(* CoDeSys 2.3.9.48 project: RCS_FB-20170118.pro *)
(* Libraries: WagoLibTerminalDiag.lib 8.11.10 11:37:48, C:\Program Files (x86)\WAGO Software\CoDeSys V2.3\Targets\WAGO\Libraries\32_Bit\SysLibMem.lib 8.11.10 11:37:48, C:\Program Files (x86)\WAGO Software\CoDeSys V2.3\Targets\WAGO\Libraries\32_Bit\SysLibRtc.lib 8.11.10 11:37:48, Util.lib 26.9.14 10:12:46, C:\Program Files (x86)\WAGO Software\CoDeSys V2.3\Targets\WAGO\Libraries\Application\WagoLib_CAN_Gateway_02.lib 25.11.15 11:32:40, C:\Program Files (x86)\WAGO Software\CoDeSys V2.3\Targets\WAGO\Libraries\Application\WagoLibMBX_System_01.lib 22.10.13 15:28:54, C:\Program Files (x86)\WAGO Software\CoDeSys V2.3\Targets\WAGO\Libraries\Application\WagoLibMBX_01.lib 20.3.12 15:32:38, Standard.lib 8.11.10 11:37:48, SYSLIBCALLBACK.LIB 8.11.10 11:37:48, WagoLibModbus_IP_01.lib 12.2.16 10:20:24, SysLibSockets.lib 5.5.11 08:22:24, Wago_MBCFG_ETHERNET_01.lib 1.4.15 13:24:28, Wago_MBCFG_COMMON_01.lib 1.4.15 13:24:28 *)

(* PLC configuration (modules and I/O channels)
0750-0658#48 CAN Gateway (48 Bytes) [Type_33_1_Channels] node 0, in %IB106 out %QB134 {INTTypePAAssignment = PLC; INTTypeModule = plugged}
  AT %IB0 [BYTEOnB_I] First Byte of 48
  AT %QB0 [BYTEOnB_Q] First Byte of 48
0750-0658#48 CAN Gateway (48 Bytes) [Type_33_1_Channels] node 1, in %IB106 out %QB134 {INTTypePAAssignment = PLC; INTTypeModule = plugged}
  AT %IB48 [BYTEOnB_I] First Byte of 48
  AT %QB48 [BYTEOnB_Q] First Byte of 48
AT %IX48.0 [BOOLOnX_I] moving negative
AT %IX48.1 [BOOLOnX_I] moving positive
AT %IX48.2 [BOOLOnX_I] On target
AT %IX48.3 [BOOLOnX_I] busy
AT %IX48.4 [BOOLOnX_I] standstill
AT %IX48.5 [BOOLOnX_I] reference ok
AT %IX48.6 [BOOLOnX_I] error, see extended info
AT %IX48.8 [BOOLOnX_I] preset input enabled
AT %IX48.9 [BOOLOnX_I] optimize on (and Z-Input for 750-636 > FW2)
AT %IX48.10 [BOOLOnX_I] extended info on
AT %IX48.11 [BOOLOnX_I] PWM active
AT %IX48.12 [BOOLOnX_I] current control on
AT %IX48.13 [BOOLOnX_I] preset input
AT %IX48.14 [BOOLOnX_I] limit switch negative
AT %IX48.15 [BOOLOnX_I] limit switch positive
AT %IW49 [WORDOnW_I] actual position low word
AT %IX49.0 [BOOLOnX_I] over temperature warning
AT %IX49.1 [BOOLOnX_I] over temperature
AT %IX49.2 [BOOLOnX_I] overflow warning
AT %IX49.3 [BOOLOnX_I] 24V ok
AT %IX49.4 [BOOLOnX_I] overload
AT %IX49.5 [BOOLOnX_I] motion detection timeout
AT %IX49.6 [BOOLOnX_I] parameter write failed
AT %IX49.7 [BOOLOnX_I] 24VL Ok (only 750-636/000-800)
AT %IX49.8 [BOOLOnX_I] 24VM Ok (only 750-636/000-800)
AT %IW50 [WORDOnW_I] actual position high word
AT %QX48.0 [BOOLOnX_Q] move negative
AT %QX48.1 [BOOLOnX_Q] move positive
AT %QX48.2 [BOOLOnX_Q] positioning
AT %QX48.3 [BOOLOnX_Q] preset
AT %QX48.4 [BOOLOnX_Q] current control on
AT %QX48.8 [BOOLOnX_Q] preset input enable
AT %QX48.9 [BOOLOnX_Q] optimize on
AT %QX48.10 [BOOLOnX_Q] extended info on
AT %QX48.15 [BOOLOnX_Q] error quit
AT %QW49 [WORDOnW_Q] target position low word
AT %QW50 [WORDOnW_Q] target position high word
0753-0430 8 DI 24 V DC 3.0ms [Type_1_8_Channels] node 3, in %IB110 out %QB134 {INTTypePAAssignment = PLC; INTTypeModule = plugged}
  AT %IX55.0 [BOOLOnX_I] Ch_1 Digital input
  AT %IX55.1 [BOOLOnX_I] Ch_2 Digital input
  AT %IX55.2 [BOOLOnX_I] Ch_3 Digital input
  AT %IX55.3 [BOOLOnX_I] Ch_4 Digital input
  AT %IX55.4 [BOOLOnX_I] Ch_5 Digital input
  AT %IX55.5 [BOOLOnX_I] Ch_6 Digital input
  AT %IX55.6 [BOOLOnX_I] Ch_7 Digital input
  AT %IX55.7 [BOOLOnX_I] Ch_8 Digital input
  AT %IX55.8 [BOOLOnX_I] Ch_1 Digital input
  AT %IX55.9 [BOOLOnX_I] Ch_2 Digital input
  AT %IX55.10 [BOOLOnX_I] Ch_3 Digital input
  AT %IX55.11 [BOOLOnX_I] Ch_4 Digital input
  AT %IX55.12 [BOOLOnX_I] Ch_5 Digital input
  AT %IX55.13 [BOOLOnX_I] Ch_6 Digital input
  AT %IX55.14 [BOOLOnX_I] Ch_7 Digital input
  AT %IX55.15 [BOOLOnX_I] Ch_8 Digital input
  AT %IX56.0 [BOOLOnX_I] Ch_1 Digital input
  AT %IX56.1 [BOOLOnX_I] Ch_2 Digital input
  AT %IX56.2 [BOOLOnX_I] Ch_3 Digital input
  AT %IX56.3 [BOOLOnX_I] Ch_4 Digital input
  AT %IX56.4 [BOOLOnX_I] Ch_5 Digital input
  AT %IX56.5 [BOOLOnX_I] Ch_6 Digital input
  AT %IX56.6 [BOOLOnX_I] Ch_7 Digital input
  AT %IX56.7 [BOOLOnX_I] Ch_8 Digital input
  AT %IX56.8 [BOOLOnX_I] Ch_1 Digital input
  AT %IX56.9 [BOOLOnX_I] Ch_2 Digital input
  AT %IX56.10 [BOOLOnX_I] Ch_3 Digital input
  AT %IX56.11 [BOOLOnX_I] Ch_4 Digital input
  AT %IX56.12 [BOOLOnX_I] Ch_5 Digital input
  AT %IX56.13 [BOOLOnX_I] Ch_6 Digital input
  AT %IX56.14 [BOOLOnX_I] Ch_7 Digital input
  AT %IX56.15 [BOOLOnX_I] Ch_8 Digital input
0753-0530 8 DO 24 V DC 0.5A [Type_10_8_Channels] node 7, in %IB113 out %QB134 {INTTypePAAssignment = PLC; INTTypeModule = plugged}
  AT %QX67.0 [BOOLOnX_Q] Ch_1 Digital output
  AT %QX67.1 [BOOLOnX_Q] Ch_2 Digital output
  AT %QX67.2 [BOOLOnX_Q] Ch_3 Digital output
  AT %QX67.3 [BOOLOnX_Q] Ch_4 Digital output
  AT %QX67.4 [BOOLOnX_Q] Ch_5 Digital output
  AT %QX67.5 [BOOLOnX_Q] Ch_6 Digital output
  AT %QX67.6 [BOOLOnX_Q] Ch_7 Digital output
  AT %QX67.7 [BOOLOnX_Q] Ch_8 Digital output
0753-0530 8 DO 24 V DC 0.5A [Type_10_8_Channels] node 8, in %IB114 out %QB134 {INTTypePAAssignment = PLC; INTTypeModule = plugged}
  AT %QX67.8 [BOOLOnX_Q] Ch_1 Digital output
  AT %QX67.9 [BOOLOnX_Q] Ch_2 Digital output
  AT %QX67.10 [BOOLOnX_Q] Ch_3 Digital output
  AT %QX67.11 [BOOLOnX_Q] Ch_4 Digital output
  AT %QX67.12 [BOOLOnX_Q] Ch_5 Digital output
  AT %QX67.13 [BOOLOnX_Q] Ch_6 Digital output
  AT %QX67.14 [BOOLOnX_Q] Ch_7 Digital output
  AT %QX67.15 [BOOLOnX_Q] Ch_8 Digital output
0753-0530 8 DO 24 V DC 0.5A [Type_10_8_Channels] node 9, in %IB114 out %QB135 {INTTypePAAssignment = PLC; INTTypeModule = plugged}
  AT %QX68.0 [BOOLOnX_Q] Ch_1 Digital output
  AT %QX68.1 [BOOLOnX_Q] Ch_2 Digital output
  AT %QX68.2 [BOOLOnX_Q] Ch_3 Digital output
  AT %QX68.3 [BOOLOnX_Q] Ch_4 Digital output
  AT %QX68.4 [BOOLOnX_Q] Ch_5 Digital output
  AT %QX68.5 [BOOLOnX_Q] Ch_6 Digital output
  AT %QX68.6 [BOOLOnX_Q] Ch_7 Digital output
  AT %QX68.7 [BOOLOnX_Q] Ch_8 Digital output
  AT %QX68.8 [BOOLOnX_Q] Ch_1 Digital output
  AT %QX68.9 [BOOLOnX_Q] Ch_2 Digital output
  AT %QX68.10 [BOOLOnX_Q] Ch_3 Digital output
  AT %QX68.11 [BOOLOnX_Q] Ch_4 Digital output
  AT %QX68.12 [BOOLOnX_Q] Ch_5 Digital output
  AT %QX68.13 [BOOLOnX_Q] Ch_6 Digital output
  AT %QX68.14 [BOOLOnX_Q] Ch_7 Digital output
  AT %QX68.15 [BOOLOnX_Q] Ch_8 Digital output
  AT %QX69.0 [BOOLOnX_Q] Ch_1 Digital output
  AT %QX69.1 [BOOLOnX_Q] Ch_2 Digital output
  AT %QX69.2 [BOOLOnX_Q] Ch_3 Digital output
  AT %QX69.3 [BOOLOnX_Q] Ch_4 Digital output
  AT %QX69.4 [BOOLOnX_Q] Ch_5 Digital output
  AT %QX69.5 [BOOLOnX_Q] Ch_6 Digital output
  AT %QX69.6 [BOOLOnX_Q] Ch_7 Digital output
  AT %QX69.7 [BOOLOnX_Q] Ch_8 Digital output
0753-0555 4 AO 4-20mA [Type_14_4_Channels] node 12, in %IB202 out %QB230 {INTTypePAAssignment = PLC; INTTypeModule = plugged}
  AT %QW51 [WORDOnW_Q] Ch_1 Analog output
  AT %QW52 [WORDOnW_Q] Ch_2 Analog output
  AT %QW53 [WORDOnW_Q] Ch_3 Analog output
  AT %QW54 [WORDOnW_Q] Ch_4 Analog output
0753-0555 4 AO 4-20mA [Type_14_4_Channels] node 13, in %IB208 out %QB236 {INTTypePAAssignment = PLC; INTTypeModule = plugged}
  AT %QW55 [WORDOnW_Q] Ch_1 Analog output
  AT %QW56 [WORDOnW_Q] Ch_2 Analog output
  AT %QW57 [WORDOnW_Q] Ch_3 Analog output
  AT %QW58 [WORDOnW_Q] Ch_4 Analog output
0753-0555 4 AO 4-20mA [Type_14_4_Channels] node 14, in %IB208 out %QB244 {INTTypePAAssignment = PLC; INTTypeModule = plugged}
  AT %QW59 [WORDOnW_Q] Ch_1 Analog output
  AT %QW60 [WORDOnW_Q] Ch_2 Analog output
  AT %QW61 [WORDOnW_Q] Ch_3 Analog output
  AT %QW62 [WORDOnW_Q] Ch_4 Analog output
0753-0555 4 AO 4-20mA [Type_14_4_Channels] node 15, in %IB208 out %QB252 {INTTypePAAssignment = PLC; INTTypeModule = plugged}
  AT %QW63 [WORDOnW_Q] Ch_1 Analog output
  AT %QW64 [WORDOnW_Q] Ch_2 Analog output
  AT %QW65 [WORDOnW_Q] Ch_3 Analog output
  AT %QW66 [WORDOnW_Q] Ch_4 Analog output
0750-0452 2 AI 0-20mA Diff [Type_8_2_Channels] node 0, in %IB208 out %QB260 {INTTypePAAssignment = PLC; INTTypeModule = plugged}
  AT %IW51 [WORDOnW_I] Ch_1 Input word
  AT %IW52 [WORDOnW_I] Ch_2 Input word
0750-0452 2 AI 0-20mA Diff [Type_8_2_Channels] node 0, in %IB208 out %QB268 {INTTypePAAssignment = PLC; INTTypeModule = plugged}
  AT %IW53 [WORDOnW_I] Ch_1 Input word
  AT %IW54 [WORDOnW_I] Ch_2 Input word
Fieldbus variables [FB_VARS] node 1, in %IB0 out %QB0
Flag variables [FLAG_VARS] node 2, in %IB0 out %QB0
Modbus-Master [MB_MASTER] node 3, in %IB0 out %QB0
*)

(* Global variable list: Global_Variables *)
VAR_GLOBAL
	FLASHER: BOOL; (* USE IN CONTROL TRANSFER *)
	FLASHER_CTRL: BOOL;
	SafetySystemOff: BOOL; (* 2.1IN   SAFETY SYSTEM OFF   --come  from hw or modbus, output ModBus *)
	SafetyStop: BOOL; (* 2.1IN   SAFETY STOP    --come form hw *)
	StartAirPressLow: BOOL; (* 2.1IN   STARTAIR PRESS. LOW     --come from pRG *)
	BR_CTRL: BOOL; (* 2.1IN   BR CTRL   come from CAN  --output  ModBus *)
	ShaftLockingDeviceEngaged: BOOL; (* 2.1IN   SHAFT LOKING DEVICE ENGAGED BX  --come from CAN *)
	StartAirValueManClosedBX: BOOL; (* 2.1IN   START AIR VALVE MAN. CLOSED BX  come from CAN  --output ModBUS *)
	SlowTurnFailBX: BOOL; (* 2.1IN     SLOW TURN. FAIL BX   --come from CAN *)
	TurningGearDiseng: BOOL; (* 2.1IN   TURNING GEAR DISENG. BX   --come from CAN *)
	ExhaustStartInterlock: BOOL; (* 2.1IN    EXHAUST VENTING START INTERLOCK --no use----only applicable for DF engine *)
	PlantInterlock: BOOL; (* 2.1IN   PLANT INTERLOCK      come from HW   --output ModBUS *)

	MVL_POS_STOP: BOOL; (* 2.1IN   MVL POSITION  STOP  --come from pRG *)
	MVL_POS_AHD_AST: BOOL; (* 2.1IN    MVL POS. AHEAD/SATERN  --come from pRG *)
	TurningGearSensorFail: BOOL; (* 2.1IN   TURNING GEAR DISENG. BX   --come from CAN *)
	EngineRun: BOOL; (* 2.1IN   ENGINE RUNNING    --come from pRG *)
	StartInterlock: BOOL; (* 2.1OUT   START REALERLOCK, PRORCS0064   --output   ModBUS *)
	H_TurnGearEngaged: BOOL; (* 2.1OUT  TURNGEARENGAGED  --output   ModBUS *)
	HornStartInterlock: BOOL; (* 2.1OUT   HORN_START_REALERLOCK   --output   PRG *)
	H_StartInterlock: BOOL; (* 2.1OUT  STARTREALERLOCK: BOOL    --output   ModBUS *)
	H_TurnGearSensorFail: BOOL; (* 2.1OUT   TURNGEARSENSORFALL    --output   ModBUS *)
	H_ShtLockDevEngaged: BOOL; (* 2.1OUT  ShtLockDevEngaged: BOOL    --output   ModBus *)
	startFail: BOOL; (* 2.2IN   START FAIL    2.2   --come from CAN *)
	MVL_POS_AHD: BOOL; (* 2.2IN   MVL POSITION AHEAD ---come from pRG---- *)
	MVL_POS_AST: BOOL := FALSE; (* 2.2IN    MVL POSITION ASTERN   ----come from pRG---- *)
	EngineStandstill: BOOL; (* 2.2IN   ENGINE STANDSTILL(STOPPED) ---come from pRG--- *)
	NNstart: BOOL; (* 2.2IN   N>NSTART   2.2--come from pRG-- *)
	EngTurnINCRSPDir: BOOL; (* IN   ENGINE TURN IN CORRESPONDING DIR    2.2  come from pRG *)
	RemoteCtrl: BOOL; (* 2.2IN   REMOTE CTRL   2.2--come from pRG-- *)
	EngTurnINNonCRSPDir: BOOL; (* 2.2IN    ENGINE TURN IN NON-CORRESPONDING DIR    2.2---come from pRG *)
	NNBrake: BOOL; (* 2.2IN     N>NBRAKE,    2.2---come from pRG *)
	AnyAuxBlowerRun: BOOL; (* 2.2IN    ANY . AUX BLOWER RUN  2.2  --come from CAN *)
	AHEAD: BOOL; (* 2.2OUT   AHEAD  2.2  --output ModBus *)
	ASTERN: BOOL; (* 2.2OUT   ASTERN   2.2   --output CAN *)
	BRAKE: BOOL; (* 2.2OUT   BRAKE    2.2   --output PRG *)
	PRESTART: BOOL; (* 2.2OUT  PRESTART     2.2  --output swd *)
	START_BRAKE: BOOL; (* 2.2OUT   START,BRAKE  2.2  --output CAN *)
	START: BOOL; (* 2.2OUT  START  2.2   --output swd *)
	STOP: BOOL; (* 2.2OUT    STOP     2.2  --output swd *)
	AllowRestartReset: BOOL; (* 2.2OUT  ALLOW RESTART RESET   2.2  --output PRG *)
	aheadastern: BOOL; (* TEMP VAR *)
	Start_Failure_BX: BOOL;
	Start_Fail_Flash_sign: BOOL;
	SLOWTURNOK: BOOL; (* 2.3IN   SLOW TURN. OK--come from CAN   output swd *)
	POWERUP: BOOL; (* 2.3IN   POWERUP   2.3   come from pRG *)

	SlowTurningBX: BOOL; (* 2.3IN  SLOW TURNING --come from CAN *)
	SlowTurnBRPush: BOOL; (* 2.3IN  SLOW TURN. BR PUSHB. --come from swd *)
	SlowTurnECRAPush: BOOL; (* 2.3IN  SLOW TURN. ECR  AUTO PUSHB.  --come from swd *)
	ECRA_CTRL: BOOL; (* 2.3IN  ECR  AUTO  CTRL --comefrom CAN *)
	SlowTurnFailReset_BR_PU: BOOL; (* 2.3IN  SLOW TURN. FAIL RESET BR PUSHB. -- come from swd *)
	SlowTurnFailReset_ECRA_PU: BOOL; (* 2.3IN  SLOW TURN. FAIL RESET  ECR  AUT. PUSHB. --come from swd *)
	SlowTurnQuest: BOOL; (* 2.3OUT  SLOW TURN.  REQUEST  --output swd *)
	SlowTurnRequestViaMVL: BOOL; (* 2.3OUT   SLOW TURNING REQUEST from MVL, PRORCS0131 --output PRG *)
	H_SlowTurning: BOOL; (* 2.3OUT  LAMP BR ECR AUT *)
	SlowTurningFailure: BOOL; (* 2.3OUT   SAME SIGNAL TO SLOWTURNFAILBX   --come from CAN、 ModBus、swd *)
	H_SlowTurnFailReset: BOOL; (* 2.3OUT  SLOW TURN. FAIL RESET   LAMP   --output SWD *)
	SlowTurnFailResetRC: BOOL; (* 2.3OUT   SLOW TURN. FAIL RESET RC    --output CAN *)
	SlowTurnRCBX: BOOL; (* 2.3OUT   SLOW TURN. RC BX   --output CAN  SWD *)
	AIRRUN: BOOL; (* 2.4IN   AIR RUN   --output swd *)
	H_AIRRUN_BR_ECR: BOOL; (* 2.4OUT   HMI AIR RUN    --output  ModBus *)
	AIRRUN_RC_BX: BOOL; (* 2.4OUT  AIR RUN RC BX  --output CAN  SWD *)
	AuxBlowerManCTRL: BOOL; (* 2.5IN   AUX BLOWER MAN. CTRL. BX  --come from CAN *)
	AuxBlowerReselECRA_PB: BOOL; (* 2.5IN   AUX BLOWER PRSEEL. ECR AUT. PUSHB  --come from SWD *)
	AuxBlowerStop_PB: BOOL; (* 2.5IN   AUX. BLOWER STOP ECR  A UT.  PUSHB. --output swd *)
	AuxBlowerFailed: BOOL; (* 2.5IN   ALL AUX. BLOWER FAILED BX --come from CAN *)
	AuxBlower_preslct_rc_ready: BOOL; (* NOT  GLOBAL_VAL *)
	H_AuxBlowerManCTRL: BOOL; (* 2.5OP   AUX. BLOWER MAN CTRL  TO HMI --output  ModBus *)
	H_AuxBlowerPresel: BOOL; (* 2.5OP   AUX. BLOWE PRESELECTED RC BX  --output  ModBus *)
	AuxBlowerPreselectedRC: BOOL; (* 2.5OP  AUX. BLOWER PRESEL. --output CAN  SWD *)
	H_AuxBlowerFailed: BOOL; (* 2.5OP   AUX. BLOWER FAIL  --output  ModBus *)
	SAFETY_SYSTEM_OFF_FAIL: BOOL; (* 2.5  SAFETY  SYSTEM OFF   2.5  come from  HW *)
	StartLearningInPro: BOOL; (* 2.6SIN   --come from CAN *)
	H_StartLearningInPro: BOOL; (* 2.6SOUT  --output  ModBus *)
	BR_PUS_BR_CTRL: BOOL; (* 2.7I    BR PUSHB. BR CTRL  --come from HW *)
	BR_PUS_ECRA_CTRL: BOOL; (* 2.7I   BR PUSHB. ECR  AUT. CTRL --come from HW *)
	BR_PUS_ECRM_CTRL: BOOL; (* 2.7I  BR PUSHB. ECR MAN. CTRL --come from HW *)
	BR_PUS_LOC_MAN_CTRL: BOOL; (* 2.7I  BR PUSHB.LOC.MAN. CTRL --come from HW *)
	ECRA_PUS_BR_CTRL: BOOL; (* 2.7I   ECR  AUT PUSHB. BR CTRL --come from HW *)
	ECRA_PUS_ECRA_CTRL: BOOL; (* 2.7I   ECR  AUT  PUSHB. ECR  AUT. CTRL --come from HW *)
	ECRA_PUS_ECRM_CTRL: BOOL; (* 2.7I  ECR  AUT  PUSHB. ECR  AUT. CTRL --come from HW *)
	ECRA_PUS_LOC_MAN_CTRL: BOOL; (* 2.7I  ECR  AUT  PUSHB.LOC.MAN. CTRL  --come from HW *)
	BRG_BRG_CTRL_FLSH: BOOL; (* 2.7I   BR LAMP BR FLASH BX --come from CAN *)
	BRG_ECRA_CTRL_FLSH: BOOL; (* 2.7I   BR LAMP ECR. AUT.FLASH BX  --come from CAN, output ModBus *)
	BRG_ECRM_CTRL_FLSH: BOOL; (* 2.7I    BR LAMP ECR. MAN.FLASH BX  --come from CAN, output ModBus *)
	BRG_LOCAL_MAN_CTRL_FLSH: BOOL; (* 2.7I   BR LAMP LOC. MAN.FLASH BX  --come from CAN, output ModBus *)
	BR_ACCOUST_CTRL_SIGN_BX: BOOL; (* 2.7I   BR ACCOUST. CT SIGNAL BX  --come from CAN, output ModBus *)
	ECR_BRG_CTRL_FLSH: BOOL; (* 2.7I     ECR LAMP BR FLASH BX --come from CAN, output ModBus *)
	ECR_ECRA_CTRL_FLSH: BOOL; (* 2.7I   ECR LAMP ECR. AUT.FLASH BX  --come from CAN, output ModBus *)
	ECR_ECRM_CTRL_FLSH: BOOL; (* 2.7I  ECR LAMP ECR. MAN.FLASH BX  --come from CAN, output ModBus *)
	ECR_LOCAL_MAN_CTRL_FLSH: BOOL; (* 2.7I   ECR  LAMP LOC. MAN.FLASH BX  --come from CAN, output ModBus *)
	ECR_ACCOUST_CTRL_SIGN_BX: BOOL; (* 2.7I   ECR  ACCOUST. CT SIGNAL BX  --come from CAN, output ModBus *)
	ECRM_CTRL: BOOL; (* ECR  MAN. CTRL *)
	LOC_MAN_CTRL: BOOL; (* LOC MAN CTRL *)
	BR_PUS_SGNL_BR_CTRL: BOOL; (* BR CTRL BX  BR PUSHB. SIGNALS  --output CAN *)
	BR_PUS_SGNL_ECRA_CTRL: BOOL; (* ECR  AUT.  BX  BR PUSHB. SIGNALS  --output CAN *)
	BR_PUS_SGNL_ECRM_CTRL: BOOL; (* ECR  MAN.  BX  BR PUSHB. SIGNALS  --output CAN *)
	BR_PUS_SGNL_LOC_MAN_CTRL: BOOL; (* LOC.MAN. CTRL BX  BR PUSHB. SIGNALS  --output CAN *)
	ECRA_PUS_SGNL_BR_CTRL: BOOL; (* BR CTRL BX  ECR AUTO PUSHB. SIGNALS  --output CAN *)
	ECRA_PUS_SGNL_ECRA_CTRL: BOOL; (* BR CTRL BX  ECR AUTO  PUSHB. SIGNALS  --output CAN *)
	ECRA_PUS_SGNL_ECRM_CTRL: BOOL; (* BR CTRL BX  ECR AUTO  PUSHB. SIGNALS  --NO--USE--- *)
	ECRA_PUS_SGNL_LOC_MAN_CTRL: BOOL; (* BR CTRL BX  ECR AUTO PUSHB. SIGNALS  --output CAN *)
	BR_LAMPS_BR_CTRL: BOOL; (* BR CTRL BR LAMPS   --output HW *)
	BR_LAMPS_ECRA_CTRL: BOOL; (* ECR AUT. CTRL.  BR  LAMPS  --output HW *)
	BR_LAMPS_ECRM_CTRL: BOOL; (* ECR MAN. CTRL.  BR LAMPS   --output HW *)
	BR_LAMPS_LOCAL_MAN_CTRL: BOOL; (* LOC. MAN. CTRL.  BR LAMPS  --output HW *)
	BR_ACCOUST_SIGN_CTRL: BOOL; (* ACCOUST. SIGN. CTRL TRANSFER BR  --output HW *)
	ECR_LAMPS_BR_CTRL: BOOL; (* BR CTRL ECR AUT. LAMPS  --output HW *)
	ECR_LAMPS_ECRA_CTRL: BOOL; (* ECR AUT. CTRL.  ECR AUT.   LAMPS  --output HW *)
	ECR_LAMPS_ECRM_CTRL: BOOL; (* ECR MAN. CTRL.  ECR AUT.  LAMPS   --output HW *)
	ECR_LAMPS_LOCAL_MAN_CTRL: BOOL; (* LOC. MAN. CTRL.  ECR AUT.  LAMPS   --output HW *)
	ECR_ACCOUST_SIGN_CTRL: BOOL; (* ACCOUST. SIGN. CTRL TRANSFER ECR   --output HW *)
	HW_ANALOG_SPEED_RCS: INT; (* 2.8AI    new signal    come from HW *)
	eng_tripped: BOOL;
	ess_overspeed_hw_bakup: BOOL; (* 2.8        come from ModBus *)
	ess_overspeed_sw_bakup: BOOL; (* 2.8        come from ModBus *)
	ess_engine_standstill_bakup: BOOL; (* 2.8          come from ModBus *)
	ess_engine_turning_astern_bkp: BOOL; (* 2.8          come from ModBus *)
	ess_engine_turning_ahead_bkp: BOOL; (* 2.8          come from ModBus *)
	POSITION_HIGHWORD: WORD; (* From hardware analog channel,address depand on the PLC configration *)
	POSITION_LOWWORD: WORD; (* From hardware analog channel,address depand on the PLC configration *)
	ANALOG_DETECT_SPEED_RCS: REAL; (* INT; 2.8AO  RCS_SPEED2  output ModBus *)
	NPN_DETECT_SPEED_RCS: INT; (* 2.8AO   RCS_SPEED1   output ModBus *)
	RCS_SPEED_MEANSURE_VALUE: REAL; (* 2.8AO  SPEED MEASURE VALUE  output HW  ModBus *)
	OVER_SPEED: BOOL; (* 2.8OUT   OVER SPEED  output  ModBus *)
	ENG_RUNING_HRS: BOOL; (* 2.8OUT   RUNNING  HOURS  output HW  ModBus *)
	PCS_SPD_MEASURE_FAILURE: BOOL; (* 2.8OUT  PCS SPEED MEASUER FAILURE   output  HW *)
	REVOLUTION_COUNTER_PULSE: BOOL; (* Address depand on the PLC configration *)
	OVERSPEED_RCS_TEMP: BOOL; (* Address depand on the PLC configration *)
	EngTurningAHD: BOOL; (* OP ENGINE TURN. AHEAD *)
	EngTurningAST: BOOL; (* OP ENGINE TURN. ASTERN *)
	RCS_SW_overspd: BOOL; (* --2.8 OVER SPEED come from SW output PRG-- *)
	RCS_HW_overspd: BOOL; (* --2.8 OVER SPEED come from HW, output ModBus-- *)
	RCS_SPD_SENSOR_FAIL1: BOOL; (* --2.8  output ModBus *)
	RCS_SPD_SENSOR_FAIL2: BOOL; (* --2.8  output ModBus *)
	MVL_POSITION_BR: REAL; (* 2.9AI  MVL POSITION BR   come from HW *)
	MVL_POSITION_ECR: REAL; (* 2.9AI  MVL POSITION  ECR    come from HW *)
	MVL_FAIL_VALUE: REAL := 3274; (* ---------2mA------------------ *)
	MVL_STOP_VALUE: REAL := 19656; (* 2.9AI  MVL STOP VALUE--------------12mA---------------- *)
	LOAD_LIMIT_IN_GAS_MODE: BOOL; (* NO  USE *)
	LOAD_LIMIT_IN_GAS_MODE_VALUE: REAL; (* NO USE *)
	SLOW_DOWN: BOOL; (* 2.9IN SLOW DOWN VALUE come from HW *)
	MAX_VALUE: REAL; (* NO USE *)
	ConvertValue: REAL := 1638; (* ------------1mA=1638-------------- *)
	Target_Elec: REAL; (* middle var *)
	SPEED_SET_SIGNALB: REAL; (* 2.9OUT   SPEED SET SIGNAL "B"    --output PRG-- *)
	SPEED_SET_SIGNALC: REAL; (* 2.9OUT   SPEED SET SIGNAL "C"   --output PRG-- *)
	HMI_BR_ECRA_CHIEFLIMIT: BOOL; (* 2.9OUT  BR ECRA CHIEF LIMIT  output  ModBus *)
	SHAFT_GENERATOR_BREAKER: BOOL; (* 2.9OUT  SHAFT GENERATOR BREAKER   --output PRG-- *)
	MVL_BR_FAIL: BOOL; (* 2.9OUT   MVL BR FAILURE   --output PRG-- *)
	MVL_ECR_FAIL: BOOL; (* 2.9OUT  MVL ECR FAILURE  output ModBus *)
	MVL_FAILURE: BOOL; (* 2.9OUT   MVL FAILURE --output PRG-- *)
	SPEED_SET_SIGNALA: REAL := 19656; (* 2.9OUT  SPEED SET SIGNALA   --output PRG---------------------------------------AVOIDING CMD MISTAKE *)
	SPEED_SETPOINT_BX: REAL; (* 2.9OUT    SPEED SETPOINT BX   output ModBus CAN *)
	RC_HANDLE_MATCH: BOOL; (* 2.9OUT      RC HANDLE MATCH BX  output CAN *)
	BR_MVL_LEVEL: REAL; (* 2.9 *)
	ECR_MVL_LEVEL: REAL; (* 2.9 *)
	BR_MVL_RPM_CMD:REAL;
	MCR_MVL_RPM_CMD:REAL;
	WRONG_WAY_ALARM: BOOL;
	H_WRONG_WAY_ALARM: BOOL; (* ------------------------------------------------------------------------------------------------ *)
	EOT_LEVER_VAULE: INT; (* 2.10  CURRENT EOT LEVER VALUE come from PRG *)
	CA_ABOVE_LIMIT_FLAG: BOOL := FALSE; (* 2.10  crash astern above limit flag,if curren lever value >= limit(90), then set true  --come from PRG-- *)
	CRASH_REVERSE_SPEEDPROGRAMOVERRIDE: BOOL;
	CRASH_REVERSE_CANCELL_LIMITS: BOOL;
	REVERSE_ACTIVE_SIGNAL: BOOL := FALSE; (* 2.10 Active  Signal *)
	SPD_SIM_MODE_ACTIVE_FLAG: BOOL;
	StartAirPressBX: REAL; (* no15AI   START AIR PRESS.BX  come from CAN *)
	StartAirPress: REAL; (* no15AO  START AIR PRESS.  output HW *)
	H_StartAirPressLow: BOOL; (* no15BO   START AIR PRESS.LOW output  ModBus *)
	ENG_FAIL_ACOUSTIC: BOOL; (* no17BO  ENGINE START FAIL ACOUSTIC  output  Modbus *)
	ALRM_ACKSOUND_OFF_PORT: BOOL;
	ALRM_ACKSOUND_OFF_STBD: BOOL;
	ALRM_ACKSOUND_OFF_ECR: BOOL;
	ALRM_ACKSOUND_OFF_BR: BOOL;
	PORT_CTRL_EOT: BOOL;
	STBD_CTRL_EOT: BOOL;
	H_HORN_ALARM_BRG: BOOL;
	H_HORN_ALARM_ECR: BOOL;
	BR_LAMP_TEST_PB_INTERNAL: BOOL;
	ECR_LAMP_TEST_PB_INTERNAL: BOOL;
	ECR_BRIDGE_IN_CONTROL_INTERNAL: BOOL;
	ECR_ECR_AUTO_IN_CONTROL_INTERNAL: BOOL;
	PORT_LAMP_TEST_PB_INTERNAL: BOOL;
	STBD_LAMP_TEST_INDICATOR_INTERNAL: BOOL;
	STBD_LAMP_TEST_PB_INTERNAL: BOOL;
	BR_CNCL_LIMIT_LMP_INTERNAL: BOOL;
	ECR_CNCEL_LIMIT_LMP_INTERNAL: BOOL;
	BR_PORT_CNCEL_LIMIT_LMP_INTERNAL: BOOL;
	BR_STBD_CNCEL_LIMIT_LMP_INTERNAL: BOOL;
	BR_CNCEL_SPEED_PRGM_LMP_INTERNAL: BOOL;
	ECR_CNCEL_SPD_PRGM_LMP_INTERNAL: BOOL;
	BR_PORT_CNCEL_SPD_PRGM_LMP_INTERNAL: BOOL;
	BR_STBD_CNCEL_SPD_PRGM_LMP_INTERNAL: BOOL;
	SPEED_PRGM_OVERRIDE_BR: BOOL;
	SPEED_PRGM_OVERRIDE_ECA: BOOL;
	BRPOT_CNCL_SPD_PRGM_SWH: BOOL;
	BRSTBD_CNCL_SPD_PRGM_SWH: BOOL;
	CANCEL_LIMITS_BR: BOOL;
	CANCEL_LIMITS_ECRA: BOOL;
	BRPOT_CANCEL_LIMIT_SWH: BOOL;
	BRSTBD_CANCEL_LIMIT_SWH: BOOL;
	MVL_FINE_ADJUST_INCREASE_RISE:BOOL;
	MVL_FINE_ADJUST_DECREASE_RISE:BOOL;
	MVL_MOVE:BOOL;
	MVL_FINE_ADJUST_AVAILABLE:BOOL;
	FINE_ADJUST_VALUE:REAL;
	SPEED_PRGM_OVERD_BX: BOOL; (* NO16  SPEED PRGM OVERRIDE  BX *)
	CANCEL_LIMITS_BX: BOOL; (* NO16  CANCEL  LIMITS  BX *)
	SPEED_PRGM_ACTIVE_INDIC: BOOL; (* NO16  SPEED  PRGM  ACTIVE INDIC. *)
	SPEED_OVERD_INDIC_BX: BOOL; (* NO16  SPEED PRGM OVERRIDE  INDIC. *)
	ENG_OUTPUT_LIMITED_BX: BOOL; (* NO16 ENG OUTPUT LIMITED BX *)
	SETPOINT_CRITICAL_SPD_BX: BOOL; (* NO16 SETPOINT  CRITICAL  SPPED BX *)
	ENG_CRITICAL_SPD_BX: BOOL; (* NO16  ENG CRITICAL SPEED BX *)
	H_SPEED_PRGM_ACTIVE: BOOL; (* NO16  SPEED PRGM ACTIVE  TO HMI *)
	H_SPD_PRGM_OVERD: BOOL; (* NO16  SPEED PRGM OVERRIDE  TO HMI *)
	H_ENG_OUTPUT_LIMITED: BOOL; (* NO16  ENG OUTPUT  LIMITED TO HMI *)
	H_SETPOINT_CRITICAL_SPD_BX: BOOL; (* NO16  SETPOINT  CRITICAL  SPEED TO HMI *)
	H_ENG_CRITICAL_SPD_BX: BOOL; (* NO16 ENG  CRITICAL  SPEED  TO  HMI *)
	propulsion_ctrl_passive_failure_alm: BOOL; (* PROPULSION CONTROL PASSIVE  FAILURE ALARM *)
	propulsion_ctrl_failure_alm: BOOL; (* PROPULSION CONTROL FAILURE ALARM *)
	PCS_POWER_SUPPLY_ALM: BOOL; (* PCS  POWER  SUPPLY  ALM *)
	ess_can_communicationLost: BOOL; (* ESS CAN COMMUNICATION *)
	BR_ECR_PUBSH_ALARM_TEST: BOOL;
	OUTPUT_LIMIT_FLASHER: BOOL; (* UNIC BACK *)
	SPEED_PRO_FLASHER: BOOL; (* UNIC BACK *)
	SPEED_AO_MAX: REAL := 32767; (* SPEED TO WATCH *)
	SPEED_AO_MIN: REAL := 0; (* SPEED TO WATCH *)
	CANIN1 AT %IB0 : ARRAY [0..47] OF BYTE;
	CANOUT1 AT %QB0 : ARRAY [0..47] OF BYTE;
	CANIN2 AT %IB48 : ARRAY [0..47] OF BYTE;
	CANOUT2 AT %QB48 : ARRAY [0..47] OF BYTE;
	Status: BYTE := 16#05;
	CANIN: ARRAY [0..17] OF BYTE;
	CANopenModbus AT %QW1000 : ARRAY [1..219] OF WORD;
	BreakDownCAN1: BOOL;
	BreakDownCAN2: BOOL;
	CommunicationLost: BOOL; (* both CAN lines are in break *)
	ByteDataFromCAN: ARRAY [0..47] OF BYTE;
	Estimated_Engine_Load_Internal: REAL; (* CAN *)
	Fuel_Index_can: REAL; (* CAN *)
	HW_ANALOG_SPEED_RCS_HW AT %IW54 : WORD; (* PRORCST5101C   AI *)
	RCS_Engine_Speed1A_HIG AT %IW50 : WORD; (* PRORCST5102C    AI *)
	RCS_Engine_Speed1B_LOW AT %IW49 : WORD; (* PRORCST5103C   AI *)
	BR_MVL_COMMD AT %IW51 : WORD; (* PRORCS1001   AI *)
	ECR_MVL_COMMD AT %IW52 : WORD; (* PRORCS1002   AI *)
	BR_ENGINE_SPEED_METER1: WORD; (* PRORCS1003    AO *)
	BR_ENGINE_SPEED_METER2: WORD; (* PRORCS1004    AO *)
	BR_ENGINE_SPEED_METER3: WORD; (* PRORCS1005    AO *)
	BR_ENGINE_SPEED_METER: WORD; (* PRORCS1006    AO *)
	BR_PORT_WING_ENGINE_SPEED_METER: WORD; (* PRORCS1007  AO *)
	BR_STBD_WING_ENGINE_SPEED_METER: WORD; (* PRORCS1008  AO *)
	CHIEF_RM_ENGINE_SPEED_METER: WORD; (* PRORCS1009  AO *)
	BR_START_AIR_PRESS_METER: WORD; (* PRORCS1010  AO *)
	BR_PORT_WING_START_AIR_PRESS_METER: WORD; (* PRORCS1011  AO *)
	BR_STBD_WING_START_AIR_PRESS_METER: WORD; (* PRORCS1012  AO *)
	ECR_START_AIR_PRESS_METER: WORD; (* PRORCS1013  AO *)
	FUEL_LOAD_INDEX: WORD; (* PRORCS1055    AO *)
	RCS_OVERSPEED_HW AT %IX55.0 : BOOL; (* PRORCS1014  DI *)
	BR_BRIDGE_APPLY_FOR_CONTROL AT %IX55.1 : BOOL; (* PRORCS1015   DI *)
	BR_ECR_AUTO_APPLY_FOR_CONTROL AT %IX55.2 : BOOL; (* PRORCS1016   DI *)
	BR_LOCAL_MAN_APPLY_FOR_CONTROL AT %IX55.3 : BOOL; (* PRORCS1017   DI *)
	BR_LAMP_TEST_PB AT %IX55.4 : BOOL; (* PRORCS1018  DI *)
	ECR_BRIDGE_APPLY_FOR_CONTROL AT %IX55.6 : BOOL; (* PRORCS1020  DI *)
	ECR_ECR_AUTO_APPLY_FOR_CONTROL AT %IX55.7 : BOOL; (* PRORCS1021  DI *)
	ECR_LOCAL_MAN_APPLY_FOR_CONTROL AT %IX55.8 : BOOL; (* PRORCS1022  DI *)
	PLANT_REALERLOCK AT %IX55.9 : BOOL; (* PRORCS1023  DI *)
	ECR_LAMP_TEST_PB AT %IX55.10 : BOOL; (* PRORCS1024  DI *)
	SAFETY_STOP AT %IX55.12 : BOOL; (* PRORCS1026   DI *)
	SAFETY_SYSTEM_OFF_HW AT %IX55.13 : BOOL; (* PRORCS1027   DI *)
	PORT_LAMP_TEST_PB: BOOL; (* PRORCS1028   DI *)
	STBD_LAMP_TEST_PB: BOOL; (* PRORCS1030  DI *)
	PCS_POWER_SUPPLY_ALM_HW AT %IX55.5 : BOOL; (* PRORCS1041  DI *)
	BR_CANCEL_LIMIT_SWH_HW AT %IX56.2 : BOOL; (* PRORCS1057    DI *)
	BR_CNCL_SPD_PRGM_SWH_HW AT %IX56.3 : BOOL; (* PRORCS1058   DI *)
	ECRA_CANCEL_LIMIT_SWH_HW AT %IX56.12 : BOOL; (* PRORCS1059    DI *)
	ECRA_CNCL_SPD_PRGM_SWH_HW AT %IX56.13 : BOOL; (* PRORCS1060   DI *)
	BRPOT_CANCEL_LIMIT_SWH_HW: BOOL; (* PRORCS1061   DI *)
	BRPOT_CNCL_SPD_PRGM_SWH_HW: BOOL; (* PRORCS1062   DI *)
	BRSTBD_CANCEL_LIMIT_SWH_HW: BOOL; (* PRORCS1063   DI *)
	BRSTBD_CNCL_SPD_PRGM_SWH_HW: BOOL; (* PRORCS1064   DI *)
	PORT_CTRL_EOT_HW: BOOL; (* PRORCS1076   DI *)
	STBD_CTRL_EOT_HW: BOOL; (* PRORCS1077   DI *)
	ESS_ENG_TURN_AHD_BKP_HW AT %IX56.6 : BOOL; (* PRORCS1078   DI *)
	ESS_ENG_TURN_AST_BKP_HW AT %IX56.7 : BOOL; (* PRORCS1079    DI *)
	SLOW_DOWN_HW AT %IX55.14 : BOOL; (* PRORCS1080   DI *)
	SAFETY_SYSTEM_OFF_FAIL_HW: BOOL; (* PRORCS1085  DI *)
	BR_BRIDGE_IN_CONTROL AT %QX67.0 : BOOL; (* PRORCS1032    DO *)
	BR_ECR_AUTO_MAN_IN_CONTROL AT %QX67.1 : BOOL; (* PRORCS1033   DO *)
	BR_LOCAL_MAN_IN_CONTROL AT %QX67.2 : BOOL; (* PRORCS1034   DO *)
	BR_LAMP_TEST_INDICATOR AT %QX67.3 : BOOL; (* PRORCS1035    DO *)
	ECR_BRIDGE_IN_CONTROL AT %QX67.6 : BOOL; (* PRORCS1038    DO *)
	ECR_ECR_AUTO_IN_CONTROL AT %QX67.7 : BOOL; (* PRORCS1039   DO *)
	ECR_LOCAL_MAN_IN_CONTROL AT %QX67.8 : BOOL; (* PRORCS1040  DO *)
	ECT_LAMP_TEST_INDICATOR AT %QX67.10 : BOOL; (* PRORCS1042    DO *)
	REVOLUTION_COUNTER_INDICATOR AT %QX67.13 : BOOL; (* PRORCS1045   DO *)
	ECR_BRIDGE_IN_CONTROL_EOT AT %QX67.15 : BOOL; (* PRORCS1047   DO *)
	ECR_ECR_AUTO_IN_CONTROL_EOT AT %QX68.0 : BOOL; (* PRORCS1048   DO *)
	PORT_LAMP_TEST_INDICATOR: BOOL; (* PRORCS1049   DO *)
	STBD_LAMP_TEST_INDICATOR: BOOL; (* PRORCS1052   DO *)
	Propulsion_Control_Failure_ALM AT %QX68.8 : BOOL; (* PRORCXS9001A   DO *)
	Propulsion_Control_Passive_Failure_ALM AT %QX68.9 : BOOL; (* PRORCXS9002A   DO *)
	PCS_ENG_Speed_Meas_Failure_ALM AT %QX68.10 : BOOL; (* PRORCXS9003A   DO *)
	Engine_Standstill_RUN_STOPPED AT %QX68.11 : BOOL; (* PRORCXS9005A   DO *)
	RUNNING_HOUR_INIDICATOR AT %QX68.7 : BOOL; (* PRORCS1056  FO *)
	BR_CNCEL_LIMIT_LMP_HW AT %QX68.14 : BOOL; (* PRORCS1065   DO *)
	BR_CNCEL_SPEED_PRGM_LMP_HW AT %QX68.15 : BOOL; (* PRORCS1066   DO *)
	ECR_CNCEL_LIMIT_LMP_HW AT %QX69.0 : BOOL; (* PRORCS1067   DO *)
	ECR_CNCEL_SPD_PRGM_LMP_HW AT %QX69.1 : BOOL; (* PRORCS1068   DO *)
	BR_PORT_CNCEL_LIMIT_LMP_HW: BOOL; (* PRORCS1069  DO *)
	BR_PORT_CNCEL_SPD_PRGM_LMP_HW: BOOL; (* PRORCS1070  DO *)
	BR_STBD_CNCEL_LIMIT_LMP_HW: BOOL; (* PRORCS1071  DO *)
	BR_STBD_CNCEL_SPD_PRGM_LMP_HW: BOOL; (* PRORCS1072  DO *)
	H_MVL_HANDLE_MATCH_mb AT %QX288.13:BOOL;   (*PRORCSMATCH  *)
	SPT_al_restar_reset_dly AT %IW256 : REAL;
	SPT_chief_limit AT %IW258 : REAL;
	SPT_crash_ast_mov_dly AT %IW260 : REAL;
	SPT_crash_ast_mvl_abv_lim AT %IW262 : REAL;
	SPT_crash_ast_mvl_bel_lim AT %IW264 : REAL;
	SPT_crash_ast_rst_spd_lim AT %IW266 : REAL;
	SPT_eng_running_dly AT %IW268 : REAL;
	SPT_engine_standstill AT %IW270 : REAL;
	SPT_fac_b_for_eng_spd AT %IW272 : REAL;
	SPT_fac_c_for_eng_spd AT %IW274 : REAL;
	SPT_flash_frequency AT %IW276 : REAL;
	SPT_lo_chief_imit AT %IW278 : REAL;
	SPT_max_speed_mb AT %IW280 : REAL; (* ----------------------------new name *)
	SPT_mvl_dslow_ahd_sp AT %IW282 : REAL;
	SPT_mvl_dslow_ast_sp AT %IW284 : REAL;
	SPT_mvl_ful_ahd_sp AT %IW286 : REAL;
	SPT_mvl_ful_sea_ahd_sp AT %IW288 : REAL;
	SPT_mvl_full_ast_sp AT %IW290 : REAL;
	SPT_mvl_full_sea_ast_sp AT %IW292 : REAL;
	SPT_mvl_half_ahd_sp AT %IW294 : REAL;
	SPT_mvl_half_ast_sp AT %IW296 : REAL;
	SPT_mvl_hand_match_thld AT %IW298 : REAL;
	SPT_mvl_posi_ahead_val AT %IW300 : REAL;
	SPT_mvl_posi_astern_val AT %IW302 : REAL;
	SPT_mvl_slow_ahd_sp AT %IW304 : REAL;
	SPT_mvl_slow_ast_sp AT %IW306 : REAL;
	SPT_mvl_stop AT %IW308 : REAL;
	SPT_n_brake_thld_hi AT %IW310 : REAL;
	SPT_n_start_thld_lo AT %IW312 : REAL;
	SPT_n_start_thld_hi AT %IW314 : REAL;
	SPT_n_brake_thld_lo AT %IW316 : REAL;
	SPT_no_gearteeth_per_rev AT %IW318 : REAL;
	SPT_rate_chan_fast AT %IW320 : REAL;
	SPT_rate_chan_low AT %IW322 : REAL;
	SPT_restar_inhibit_dly AT %IW324 : REAL;
	SPT_rev_count_factor AT %IW326 : REAL;
	SPT_slowdown_val AT %IW328 : REAL;
	SPT_slowturn_by_MVL_enab AT %IW330 : REAL;
	SPT_slowturn_del_req AT %IW332 : REAL;
	SPT_spd_CMCR AT %IW334 : REAL;
	SPT_spd_pulse_time AT %IW336 : REAL;
	SPT_star_air_pres_hi AT %IW338 : REAL;
	SPT_star_air_pres_low AT %IW340 : REAL;
	SPT_over_speed AT %IW352 : REAL;
	SPT_sim_mode_active AT %IW354 : REAL;
	SPT_speed_from_hmi AT %IW356 : REAL;
	SPT_speed_hmi AT %IW358 : REAL;
	SPT_Critical_Speed_Enable AT %IW360 : REAL;
	SPT_Critical_RPM_low1 AT %IW362 : REAL;
	SPT_Critical_RPM_high1 AT %IW364 : REAL;
	SPT_Critical_RPM_low2 AT %IW366 : REAL;
	SPT_Critical_RPM_high2 AT %IW368 : REAL;
	SPT_mvl_fine_stage AT %IW452:REAL;
	SPT_mvl_fine_max AT %IW454:REAL;
	SPT_mvl_fine_reset AT %IW456:REAL;
	ess_eng_turning_ahead_bkp_mb: BOOL; (* come from ESS:PROESS0072 *)
	ess_eng_turning_astern_bkp_mb: BOOL; (* come from ESS:PROESS0073 *)
	ess_eng_standstill_bkp_mb: BOOL; (* come from  ESS:PROESS0003 *)
	ess_eng_speed_bkp_mb: REAL; (* come from  ESS:PROESS0004 *)
	ess_overspeed_sw_bkp_mb: BOOL; (* come from  ESS:PROESS0062 *)
	ess_overspeed_hw_bkp_mb: BOOL; (* come from ESS:PROESS0075 *)
	alrm_acksound_off_br_mb: BOOL; (* come from ESS:PROESS0118 *)
	alrm_acksound_off_ecr_mb: BOOL; (* come from ESS:PROESS0119 *)
	alrm_acksound_off_port_mb: BOOL; (* come from ESS:PROESS0120 *)
	alrm_acksound_off_stbd_mb: BOOL; (* come from ESS:PROESS0121 *)
	safety_stop_mb: BOOL; (* come from ESS:PROESS0103 *)
	start_air_pressure AT %QW256 : REAL; (* PRORCCAN0001	START AIR PRESSURE *)
	eng_revolution_counter AT %QW258 : REAL; (* PRORCS0055	ENGINE REVOLUTION COUNTER   no use *)
	rcs_eng_speed1 AT %QW262 : REAL; (* PRORCS0089  	  RCS ENGINE SPEED 1 *)
	eng_speed_setpoint_rc AT %QW264 : REAL; (* PRORCS0090  	Engine speed  setpoint RC *)
	fuel_index AT %QW466 : REAL; (* PRORCS0104	Engine LOAD INDEX *)
      h_fuel_index AT %QW472 : REAL; (*PRORCS7174, FUEL INDEX*)
	slow_turning_mb AT %QX284.0 : BOOL; (* PRORCCAN1001   SLOW TURNING 	         SP_swd_perm_rcs1_1_62 *)
	slow_turnok_mb AT %QX284.1 : BOOL; (* PRORCCAN1002	SLOW TURNING OK	   SP_swd_perm_rcs1_2_62 *)
	slow_turning_failure_mb AT %QX284.2 : BOOL; (* PRORCCAN1003	SLOW TURNING FAIL. 	SlowTurningFailure  Slow_Turning_Failure_mb	SP_swd_perm_rcs1_3_62 *)
	start_failure_alm AT %QX284.3 : BOOL; (* PRORCCAN1004     START FAILURE Alarm     SP_swd_perm_rcs1_4_62 *)
	start_air_valve_man_closed AT %QX284.4 : BOOL; (* PRORCCAN1005    START AIR VALVE MAN. CLOSED	       SP_swd_perm_rcs1_5_62 *)
	turning_gear_engaged_alm AT %QX284.5 : BOOL; (* PRORCCAN1006   TURNING GEAR ENGAGED   Alarm    SP_swd_perm_rcs1_6_62 *)
	turning_gear_sensor_failure_alm AT %QX284.6 : BOOL; (* PRORCCAN1007  TURNING GEAR SENSOR FAILURE   Alarm     SP_swd_perm_rcs1_7_62 *)
	any_aux_blower_run_mb AT %QX284.7 : BOOL; (* PRORCCAN1008	ANY AUX. BLOWER RUNNING          	SP_swd_perm_rcs1_8_62 *)
	aux_blower_manctrl_mb AT %QX284.8 : BOOL; (* PRORCCAN1009	AUXILIARY BLOWER MANUAL CONTROL INDICA.     SP_swd_perm_rcs1_9_62 *)
	aux_blower_failed_mb AT %QX284.9 : BOOL; (* PRORCCAN1010	     ALL AUX. BLOWERS FAILED	   SP_swd_perm_rcs1_10_62 *)
	speed_prgm_override AT %QX284.10 : BOOL; (* PRORCCAN1011    SPEED PRGM. OVERRIDE 	   SP_swd_perm_rcs1_11_62 *)
	eng_output_limited AT %QX284.11 : BOOL; (* PRORCCAN1012    ENGINE OUTPUT LIMITED         SP_swd_perm_rcs1_12_62 *)
	setpoint_critical_speed AT %QX284.12 : BOOL; (* PRORCCAN1013   SETPOINT CRITICAL SPEED     SP_swd_perm_rcs1_13_62 *)
	eng_critical_speed AT %QX284.13 : BOOL; (* PRORCCAN1014   ENGINE CRITICAL SPEED         SP_swd_perm_rcs1_14_62 *)
	unic_start_learning_inprogress_indica AT %QX284.14 : BOOL; (* PRORCCAN1015   START LEARNING IN PROGRESS INDICA.  SP_swd_perm_rcs1_15_62 *)
	speed_prgm_active AT %QX284.15 : BOOL; (* PRORCCAN1016   SPEED PRGM. ACTIVE     SP_swd_perm_rcs1_16_62 *)
	bridge_ctrl AT %QX285.0 : BOOL; (* PRORCCAN2001     BRIDGE CONTROL	          SP_swd_perm_rcs2_1_62 *)
	ecr_aut_ctrl AT %QX285.1 : BOOL; (* PRORCCAN2002    ECR AUTOM. CONTROL    SP_swd_perm_rcs2_2_62 *)
	ecr_man_ctrl AT %QX285.2 : BOOL; (* PRORCCAN2003   ECR MAN. CONTROL  	 SP_swd_perm_rcs2_3_62 *)
	local_man_ctrl AT %QX285.3 : BOOL; (* PRORCCAN2004   LOCAL MAN. CONTROL   SP_swd_perm_rcs2_4_62 *)
	br_lamp_br_flash AT %QX285.4 : BOOL; (* PRORCCAN2005	BRIDGE LAMP “BRIDGE” FLASH   SP_swd_perm_rcs2_5_62 *)
	br_lamp_ecr_autom_flash AT %QX285.5 : BOOL; (* PRORCCAN2006      BRIDGE LAMP “ECR AUTOM.” FLASH	  SP_swd_perm_rcs2_6_62 *)
	br_lamp_ecr_man_flash AT %QX285.6 : BOOL; (* PRORCCAN2007      BRIDGE LAMP “ECR MAN.” FLASH	         SP_swd_perm_rcs2_7_62 *)
	br_lamp_local_man_flash AT %QX285.7 : BOOL; (* PRORCCAN2008      BRIDGE LAMP “LOCAL MAN.” FLASH          SP_swd_perm_rcs2_8_62 *)
	br_accoustic_ctrl_transfer_signal AT %QX285.8 : BOOL; (* PRORCCAN2009	    BRIDGE ACCOUSTIC CONTROL TRANSFER SIGNAL	 SP_swd_perm_rcs2_9_62 *)
	ecr_lamp_br_flash AT %QX285.9 : BOOL; (* PRORCCAN2010	     ECR   LAMP “BRIDGE” FLASH      SP_swd_perm_rcs2_10_62 *)
	ecr_lamp_ecr_autom_flash AT %QX285.10 : BOOL; (* PRORCCAN2011	   ECR LAMP “ECR AUTOM.” FLASH	   SP_swd_perm_rcs2_11_62 *)
	ecr_lamp_ecr_man_flash AT %QX285.11 : BOOL; (* PRORCCAN2012 	   ECR LAMP “ECR MAN.” FLASH	          SP_swd_perm_rcs2_12_62 *)
	ecr_lamp_local_man_flash AT %QX285.12 : BOOL; (* PRORCCAN2013    ECR LAMP “LOCAL MAN.” FLASH      SP_swd_perm_rcs2_13_62 *)
	ecr_ccoustic_ctrl_transfer_signal AT %QX285.13 : BOOL; (* PRORCCAN2014	ECR ACCOUSTIC CONTROL TRANSFER SIGNAL	SP_swd_perm_rcs2_14_62 *)
	shaft_locking_dev_engaged AT %QX285.14 : BOOL; (* PRORCCAN2015	  shaft_locking_dev_engaged      SP_swd_perm_rcs2_15_62 *)
	over_speed_rcs_mb AT %QX286.0 : BOOL; (* PRORCS0001	RCS OVERSPEED BKP		SP_swd_perm_rcs3_1_62 *)
	rcs_overspeed_sw AT %QX286.1 : BOOL; (* PRORCS0047	RCS OVERSPEED SW	rcs_overspeed_sw  	SP_swd_perm_rcs3_2_62 *)
	rcs_overspeed_hw_mb AT %QX286.2 : BOOL; (* PRORCS0048   RCS OVERSPEED HW      SP_swd_perm_rcs3_3_62 *)
	air_run_indicator AT %QX286.3 : BOOL; (* PRORCS0049	AIR RUN INDICATOR	  	SP_swd_perm_rcs3_4_62 *)
	rcs_mvl_br_failure AT %QX286.4 : BOOL; (* PRORCS0050	RCS MVL BR FAILURE	 SP_swd_perm_rcs3_5_62 *)
	rcs_mvl_ecr_failure AT %QX286.5 : BOOL; (* PRORCS0051	RCS MVL ECR FAILURE	  	SP_swd_perm_rcs3_6_62 *)
	aux_blower_preselecRC_mb AT %QX286.6 : BOOL; (* PRORCS0052  	AUXILIARY BLOWER PRESELECTED INDICATOR	    SP_swd_perm_rcs3_7_62 *)
	chief_limit_speed_indicaotr AT %QX286.7 : BOOL; (* PRORCS0057	CHIEF LIMIT  SPEED INDICAOTRSP_swd_perm_rcs3_8_62 *)
	rcs_eng_speed_sensor1_failure AT %QX286.8 : BOOL; (* PRORCS0058	RCS ENGINE SPEED 1 FAILURE	SP_swd_perm_rcs3_9_62 *)
	rcs_eng_speed_sensor2_failure AT %QX286.9 : BOOL; (* PRORCS0059	RCS ENGINE GRP SPEED 2 FAILURE	SP_swd_perm_rcs3_10_62 *)
	startair_press_low_alm AT %QX286.10 : BOOL; (* PRORCS0063	STARTAIR PRESS. LOW ALARM 	  SP_swd_perm_rcs3_11_62 *)
	start_interlock_alm AT %QX286.11 : BOOL; (* PRORCS0064	START INTERLOCK  ALARM 	  SP_swd_perm_rcs3_12_62 *)
	propulsion_ctrl_failure_alm_mb AT %QX286.12 : BOOL; (* PRORCS0069 Propulsion Control Failure ALM.   SP_swd_perm_rcs3_13_62 *)
	propulsion_ctrl_passive_failure_alm_mb AT %QX286.13 : BOOL; (* PRORCS0070 Propulsion Control Passive Failure ALM.	  SP_swd_perm_rcs3_14_62 *)
	propulsion_ctrl_speed_meas_failure_alm AT %QX286.14 : BOOL; (* PRORCS0071	Propulsion Control Speed Meas. Failure ALM.	SP_swd_perm_rcs3_15_62 *)
	rcs_comm_to_unic_lost_failure AT %QX287.0 : BOOL; (* PRORCS0072	RCS COMM TO UNIC LOST FAILURE  SP_swd_perm_rcs4_1_62 *)
	rcs_can1_TO_unic_lost_failure AT %QX287.1 : BOOL; (* PRORCS0073	RCS CAN1 TO UNIC LOST FAILURE	  SP_swd_perm_rcs4_2_62 *)
	rcs_can2_to_unic_lost_failure AT %QX287.2 : BOOL; (* PRORCS0074	RCS CAN2 TO UNIC LOST FAILURE	  SP_swd_perm_rcs4_3_62 *)
	eng_starting AT %QX287.3 : BOOL; (* PRORCS0075  ENGINE STARTING  SP_swd_perm_rcs4_4_62 *)
	eng_running AT %QX287.4 : BOOL; (* PRORCS0076	 ENGINE RUNNING  	SP_swd_perm_rcs4_5_62 *)
	eng_ready_for_start AT %QX287.5 : BOOL; (* PRORCS0077	ENGINE READY for START 	SP_swd_perm_rcs4_6_62 *)
	eng_not_ready AT %QX287.6 : BOOL; (* PRORCS0078	ENGINE NOT READY	  SP_swd_perm_rcs4_7_62 *)
	eng_stopping AT %QX287.7 : BOOL; (* PRORCS0079	ENGINE STOPPING  	SP_swd_perm_rcs4_8_62 *)
	eng_stopped AT %QX287.8 : BOOL; (* PRORCS0080 	ENGINE STOPPED	SP_swd_perm_rcs4_9_62 *)
	rcs_eng_speed2 AT %QW360 : REAL; (* PRORCS0081	RCS ENGINE SPEED 2 	 SP_swd_perm_rcs4_9_62 *)
	safety_system_off AT %QX287.10 : BOOL; (* PRORCS0082	SAFETY SYSTEM OFF      SP_swd_perm_rcs4_11_62 *)
	eng_tripped_mb AT %QX287.11 : BOOL; (* PRORCS0083	ENGINE TRIPPED 	 SP_swd_perm_rcs4_12_62 *)
	mvl_postion_ahead AT %QX287.12 : BOOL; (* PRORCS0091	MVL POSTION= AHEAD   	SP_swd_perm_rcs4_13_62 *)
	mvl_postion_astern AT %QX287.13 : BOOL; (* PRORCS0092	MVL POSTION= ASTERN    SP_swd_perm_rcs4_14_62 *)
	mvl_postion_stop AT %QX287.14 : BOOL; (* PRORCS0093     MVL POSTION= STOP  SP_swd_perm_rcs4_15_62 *)
	ahead_cmd AT %QX288.0 : BOOL; (* PRORCS0094    AHEAD CMD	  SP_swd_perm_rcs5_1_62 *)
	astern_cmd AT %QX288.1 : BOOL; (* PRORCS0095	ASTERN CMD	  	SP_swd_perm_rcs5_2_62 *)
	stop_cmd AT %QX288.2 : BOOL; (* PRORCS0096	STOP CMD	SP_swd_perm_rcs5_3_62 *)
	rcs_eng_turning_ahead AT %QX288.3 : BOOL; (* PRORCS0099	RCS ENGINE TURNING AHEAD	      SP_swd_perm_rcs5_4_62 *)
	rcs_eng_turning_astern AT %QX288.4 : BOOL; (* PRORCS0100	RCS ENGINE TURNING ASTERN 	SP_swd_perm_rcs5_5_62 *)
	pcs_system_ready AT %QX288.5 : BOOL; (* PRORCS0103	 PCS SYSTEM READY	  SP_swd_perm_rcs5_6_62 *)
	plant_interlock AT %QX288.6 : BOOL; (* PRORCS0107	PLANT INTERLOCK     	SP_swd_perm_rcs5_7_62 *)
	remote_ctrl_failure AT %QX288.7 : BOOL; (* PRORCS0108	REMOTE CONTROL FAILURE   	SP_swd_perm_rcs5_8_62 *)
	safety_sys_stop_mb AT %QX288.8 : BOOL; (* PRORCS9004    SP_swd_perm_rcs5_9_62 *)
	ecr_lamp_test_pb_mb AT %QX288.9 : BOOL; (* PRORCS0139	ECR LAMP TEST PB.     SP_swd_perm_rcs5_10_62 *)
	br_lamp_test_pb_mb AT %QX288.10 : BOOL; (* PRORCS0140 	BR LAMP TEST PB.      SP_swd_perm_rcs5_11_62 *)
	br_portlamp_test_pb_mb AT %QX288.11 : BOOL; (* PRORCS0141	PORT LAMP TEST PB.     SP_swd_perm_rcs5_12_62 *)
	br_stbdlamp_test_pb_mb AT %QX288.12 : BOOL; (* PRORCS0142	STBD LAMP TEST PB.     SP_swd_perm_rcs5_13_62 *)
	spd_sim_mode_active_mb AT %QX289.11 : BOOL; (* PRORCS0157	 Speed simulation mode Active        SP_swd_perm_rcs6_12_62 *)
	startfail_horn_alm_mb AT %QX289.12 : BOOL; (* PRORCS0158   	StartFail HORN ALARM		SP_swd_perm_rcs6_13_62 *)
	horn_alarm_mb AT %QX289.13 : BOOL; (* PRORCS0164	HORN SPEAKER	horn_alarm_mb	SP_swd_perm_rcs6_14_62 *)
	h_horn_alarm_brg_mb AT %QX389.14 : BOOL;
	h_horn_alarm_mcr_mb AT %QX389.15 : BOOL;
	port_ctrl_rc_es AT %QX287.9 : BOOL; (* PRORCS9001 *)
	stbd_ctrl_rc_es AT %QX287.15 : BOOL; (* PRORCS9002 *)
	rcs_speed_meansure_value_mb AT %QW362 : REAL; (* PRORCS9003 *)
	br_mvl_level_mb AT %QW370 : REAL;
	ecr_mvl_level_mb AT %QW372 : REAL;
	br_ecr_pubsh_alarm_test_mb: BOOL; (* new signal ------------------------------ *)
	SWD_swd_me_62 AT %QW268 : UINT;
	SWD_swd_cont_position_0 AT %QW270 : UINT;
	SWD_swd_oper_mode_62 AT %QW272 : UINT;
	SC_swd_oper_mode_62 AT %IW343 : UINT;
	SCS_swd_oper_mode_1_62 AT %QW273 : UINT;
	SCS_swd_oper_mode_2_62 AT %QW274 : UINT;
	SWD_swd_mvl_direct_0 AT %QW275 : UINT;
	SWD_swd_aux_blower_62 AT %QW276 : UINT;
	SC_swd_aux_blower_62 AT %IW344 : UINT;
	SCS_swd_aux_blower_1_62 AT %QW277 : UINT;
	SCS_swd_aux_blower_2_62 AT %QW278 : UINT;
	SWD_swd_slow_turn_62 AT %QW279 : UINT;
	SC_swd_slow_turn_62 AT %IW345 : UINT;
	SCS_swd_slow_turn_1_62 AT %QW280 : UINT;
	SCS_swd_slow_turn_6_62 AT %QW281 : UINT;
	SWD_swd_air_run_62 AT %QW282 : UINT;
	(*SC_swd_air_run_62 AT %IW346 : UINT;*)
      CP_BUTAIRRUN AT %IW346: REAL;
      PERAIRRUN AT %QX283.1: BOOL;
      SWD_swd_merpmlim_0 AT %QW474: UINT;
	(*SCS_swd_air_run_1_62 AT %QW283 : UINT;*)
	h_br_mvl_rpm_cmd_mb AT %QW468:REAL;(*PROBRGCMDRPM*)
	h_ecr_mvl_rpm_cmd_mb AT %QW470:REAL;(*PROMCRCMDRPM*)
	h_speed_cmd_adjust_mb AT %IW350:REAL;(*--------1-INCREASE,      0-NO ACTION,       -1-DECREASE-----------*)
END_VAR
VAR_GLOBAL RETAIN
	SPEED_CMCR: REAL; (* NO USE---------------------------------------------------------------NO USE-- *)
	SPD_SIM_MODE_ACTIVE: REAL;
	GRADE_RPM_ELEC_MAP: ARRAY [0..10] OF POINTS := (GRADE := 0,RPM:=102,ELEC:=32760),
(GRADE := 1,RPM:=99,ELEC:=31122),(GRADE := 2,RPM:=49,ELEC:=29484),(GRADE := 3,RPM:=44,ELEC:=26208),
(GRADE := 4,RPM:=39,ELEC:=22932),(GRADE :=5,RPM:=0,ELEC:=19656),(GRADE := 6,RPM:=39,ELEC:=16380),
(GRADE := 7,RPM:=44,ELEC:=13104),(GRADE := 8,RPM:=49,ELEC:=9828),(GRADE := 9,RPM:=69,ELEC:=8190),
(GRADE := 10,RPM:=84,ELEC:=6552); (* --output PRG-- *)
	SIMULATION_TARGET_VALUE: REAL;
	SIMULATION_TARGET_VALUE_FROMHMI: REAL;
	SMI_SPD_FROM_HMI: REAL;
	OVERSPEED_SETPOINT: INT; (* 2.8  OVER SPEED SETPOINT come from ModBus; *)
	StartAirPreLow: REAL; (* no15AI  THRESHOLDS LOW come from ModBus *)
	StartAirPreHIGH: REAL; (* no15AI PRESS. THRESHOLDS HIGH come from ModBus *)
	PULSE_TIME: TIME; (* 2.9TI   PULSE TIME   comefrom ModBus *)
	SlowTurnDelayRequest: TIME; (* 2.3DI SLOW TURN DELAY OF REQUEST--come from ModBus *)
	SlowByMVLEnable: BOOL; (* 2.3DI  SLOW BY MVL ENABLE --come from ModBus *)
	SLOW_DOWN_VALUE: REAL; (* 2.9AI  SLOW DOWN VALUE come from ModBus *)
	REVOLUTION_COUNTER_FACTOR_SETPOINT: INT; (* 2.8AI     REV. COUNTER     come from ModBus *)
	RstartInhibitDelay: TIME; (* 2.2DI    RESTART INHIBIT DELAY   2.2   come from ModBus *)
	RATE_OF_CHANGE_SLOW: REAL; (* 2.9AI  RATE OF CHANGE SLOW   come from ModBus *)
	RATE_OF_CHANGE_FAST: REAL; (* 2.9AI  RATR OF CHANGE FAST    come from ModBus *)
	GEAR_TEETH_PER_REVOLUTION_SETPOINT: INT; (* 2.8AI   NUMBER  OF  GREAR  TEETH  PER REVOLUTION:REAL; come from ModBus *)
	NBreakLOW: REAL; (* 2.12AI   THRESHOLDS   come from ModBus *)
	NStartHIGH: REAL; (* 2.12AI   THRESHOLDS     come from ModBus *)
	NStartLOW: REAL; (* 2.12AI   THRESHOLDS      come from ModBus *)
	NBreakHIGH: REAL; (* 2.12AI  THRESHOLDS   come from ModBus *)
	MVL_POS_ASTERN_VALUE: REAL; (* 2.9AI MVL POS ASTERN VALUE  come from ModBus *)
	MVL_POS_AHEAD_VALUE: REAL; (* 2.9AI  MVL POS AHEAD VALUE  come from ModBus *)
	MVL_HANDLE_MATCH: REAL; (* 2.9 MVL HANDLE MATCH  come from ModBus *)
	MAX_SPEED: REAL; (* 2.9AI  MAX. SPEED  come from ModBus *)
	LO_CHIEF_LIMIT: REAL; (* 2.9AI LO CHIEF LIMIT   come from  ModBus *)
	HZ: REAL := 1.0;
	SPEED_FACTOR_C: REAL; (* 2.8AI    come from ModBus *)
	SPEED_FACTOR_B: REAL; (* 2.8AI    come from ModBus *)
	STANDSTILL_SETPOINT: INT; (* 2.8AI   ENG  STANDSTILL   come from ModBus *)
	EngineRuningDelay: TIME; (* no14AI  ENGINE RUN. DELAY  come from ModBus *)
	REAL_Crash_Astern_S3: REAL := -60; (* 2.10     Reset Creash Astern above This  Limit    --come from ModBus *)
	Activate_Crash_Astern_S2: REAL := -85; (* 2.10  Active Creash Astern below This Limit   --come from ModBus *)
	Enable_Crash_Astern_S1: REAL := 90; (* 2.10   Enable  Crash  Astern  Above This Limit  --come from ModBus *)
	CrashMovDly: TIME; (* 2.10  Lever move time   --come from ModBus *)
	CHIEFLIMIT: REAL; (* 2.9AI  CHIEF LIMIT  come from ModBus *)
	AllowRestartResetDelay: TIME; (* 2.2TI     ALLOW  RESTART RESET   2.2--come from ModBus *)
	Critical_Speed_Enable: REAL;
	Critical_RPM_low1: REAL;
	Critical_RPM_high1: REAL;
	Critical_RPM_low2: REAL;
	Critical_RPM_high2: REAL;

(*CAN*)

	CANIN1_CHG_FLAG:	BOOL;
	CANIN2_CHG_FLAG:	BOOL;

END_VAR

(* Data type *)
TYPE POINTS :
STRUCT
	GRADE :REAL;
	RPM:REAL;
	ELEC:REAL;
END_STRUCT
END_TYPE

(* POU PLC_PRG, ST *)
PROGRAM PLC_PRG
VAR
    FLASHER_PRODUCER_FUNC:   Flasher_Producer;
    ME_START_PERMISSIVES_FUNC:   ME_Start_Permissives;(*---4.1.5.2.1 ME Start  Permissives--*)
    ME_START_BRAKE_SEQUENCE_FUNC:  ME_Start_Brake_Sequence;(*---4.1.5.2.2  ME Start, Break Sequence--*)
    SLOW_TURNING_SEQUENCE_FUNC:  Slow_Turning_Sequence;(*---4.1.5.2.3 SLOW TURNING SEQUENCE--*)
    AIR_RUN_SEQUENCE_FUNC:  Air_Run_Sequence;(*---4.1.5.2.4 Air Run Sequence--*)
    AUXILIARY_BLOWER_FUNC: Auxiliary_Blower;(*---4.1.5.2.5--*)
    CRANK_ANGLE_SYSTEM_FUNC:Crank_Angle_System;(*---4.1.5.2.6--*)
    CTRL_TRANSFER_FUNC:  Control_Transfer;(*-----------------4.1.5.2.7 CTRL  TRANSFER  ------------  *)
    SPEED_CONTROL_FUNC: Speed_Control;(*---4.1.5.2.9 Speed Control--*)
    CRASH_REVERSE_FUNC: Crash_Reverse;(*---4.1.5.2.10 Crash Reverse--*)
    SIMULATION_MODE_FUNC:Simulation_Mode;(*---4.1.5.2.11 SIMULATION_MODE_FUNC--*)
(*------------------NO12  SPEED  THRESHOLDS-----------------*)
(* ---------------- NO13 ENG. TURNING IN  CORRESPONDING  NON-CORRESPONDING  DIRECTION----*)
(*------------------NO14   ENGINE  RUNNING -------------------*)
(*------------------NO15   START AIR PRESSURE-------------------------*)
	OTHER_FUNCTION_FUNC:Other_Function;

(*------NO16  ACOUSTIC    SIGNALS-------*)
	ME_OVRD_LIMIT_INST:Me_Over_Limit;

(*------------------NO17-ME OVER LIMIT------------------------------*)

(*-------------------------NO18 LAMP TEST--------------------*)
	AUX_FUNCTION_FUNC:LAMP_TEST;
	LAMP_FUNCT:LAMP;
	TON_PWR_UP_FUNC:TON;
	HW_PARAM_FUNC: PARAM_HW;
	MODBUS_PARAM_FUNC:  PARAM_MODBUS;
	SWD_FUNC: SWD;
	Critical_RPM_FUNC:Critical_RPM;
	Unic_Back_FUNC:Unic_Back;

(*-----------------------CAN----------------------*)
	CANRead_FUNC:CANRead;
	CANWrite_FUNC:CANWrite;

END_VAR
(*Speed_Control_INST();*)

	TON_PWR_UP_FUNC(IN:=TRUE, PT:=T#1000ms);
 	 IF ( NOT  TON_PWR_UP_FUNC.Q) THEN
         POWERUP:=TRUE;
 	  END_IF


         (*-------initial signal---------*)

   FLASHER_PRODUCER_FUNC;

    ME_START_PERMISSIVES_FUNC;(*---4.1.5.2.1  ME Start  Permissives--*)

    ME_START_BRAKE_SEQUENCE_FUNC;(*---4.1.5.2.2   ME Start, Break Sequence--*)

    SLOW_TURNING_SEQUENCE_FUNC;(*---4.1.5.2.3  SLOW TURNING SEQUENCE--*)

    AIR_RUN_SEQUENCE_FUNC;(*---4.1.5.2.4  Air Run Sequence--*)

    AUXILIARY_BLOWER_FUNC;(*---4.1.5.2.5  AUXILIARY BLOWER--*)

    CRANK_ANGLE_SYSTEM_FUNC;(*---4.1.5.2.6 CRANK ANGLE SYSTEM--*)

    CTRL_TRANSFER_FUNC;(*---4.1.5.2.7 CTRL  TRANSFER  ---*)

    SPEED_MEASUREMENT_RCS;(*---4.1.5.2.8  SPEED  MEASUREMENT *)

    SPEED_CONTROL_FUNC;(*---4.1.5.2.9  Speed Control--*)

    CRASH_REVERSE_FUNC;(*---4.1.5.2.10  Crash Reverse--*)

    SIMULATION_MODE_FUNC;(*---4.1.5.2.11 Ship_Testbed_Mode--*)

    OTHER_FUNCTION_FUNC;

    ME_OVRD_LIMIT_INST;

    AUX_FUNCTION_FUNC;

    LAMP_FUNCT;

    TON_PWR_UP_FUNC;

    HW_PARAM_FUNC;

    MODBUS_PARAM_FUNC;

    SWD_FUNC;

   Unic_Back_FUNC;

   Critical_RPM_FUNC;

(*-----------------------CAN----------------------*)

    IF(NOT CommunicationLost)
    THEN
    CANRead_FUNC;
    CANWrite_FUNC;
    END_IF

(*---------------send buzzer signal from rcs to EOT----------------------*)
 horn_alarm_mb:=( ENG_FAIL_ACOUSTIC OR BR_ECR_PUBSH_ALARM_TEST) ;(*PRORCS0164	horn_alarm_mb	%QX289.13*)

h_horn_alarm_brg_mb:=H_HORN_ALARM_BRG;

h_horn_alarm_mcr_mb:=H_HORN_ALARM_ECR;
END_PROGRAM

(* POU Flasher_Producer, ST *)
FUNCTION_BLOCK Flasher_Producer
VAR_INPUT
END_VAR
VAR_OUTPUT
END_VAR
VAR
      FLASH_INST:  BLINK;
      FLASH_INST2: BLINK;

	timeHZ: TIME;

	HZ_INT: INT;
	temp: REAL;
	timer: REAL;
	times: TIME;
	HZ_TEMP: REAL := 1.0;
END_VAR
(*  GLOBAL_VAR   product   blinker*)



   (* timeHZ:=REAL_TO_TIME((1.0/HZ_TEMP)*0.5*1000);(*HZ come from setpoint*)*)
    IF HZ = 0.0  THEN   HZ := 1.0;    END_IF
    timeHZ:=REAL_TO_TIME((1.0/HZ)*0.5*1000);(*HZ come from setpoint*)

 FLASH_INST(ENABLE:=TRUE, TIMELOW:=timeHZ,TIMEHIGH:=timeHZ);
 FLASHER:=FLASH_INST.OUT;


IF ((ALRM_ACKSOUND_OFF_BR AND BR_CTRL)OR (ALRM_ACKSOUND_OFF_ECR AND ECRA_CTRL )OR (ALRM_ACKSOUND_OFF_PORT AND  PORT_CTRL_EOT) OR (ALRM_ACKSOUND_OFF_STBD AND STBD_CTRL_EOT ))
THEN
  FLASHER_CTRL:=TRUE;
ELSE
     FLASH_INST2(ENABLE:=TRUE, TIMELOW:=timeHZ,TIMEHIGH:=timeHZ);
     FLASHER_CTRL:=FLASH_INST2.OUT;
END_IF;
END_FUNCTION_BLOCK

(* POU ME_Start_Permissives, ST *)
FUNCTION_BLOCK ME_Start_Permissives
VAR_INPUT
END_VAR
VAR_OUTPUT
END_VAR
VAR


	Rtemp: BOOL;
	Stemp: BOOL;
	SR_FUNS: SR;
END_VAR
(*---------4.1.5.2.1 ME Start  Permissives------------*)

(* Set  StartInterlock   Value  *)
Stemp:=(SafetySystemOff
             OR SafetyStop
             OR( StartAirPressLow AND BR_CTRL)
             OR ShaftLockingDeviceEngaged
             OR StartAirValueManClosedBX
             OR SlowTurnFailBX
             OR (NOT TurningGearDiseng)
             OR ExhaustStartInterlock
             OR PlantInterlock
);
Rtemp:=MVL_POS_STOP  AND(NOT  Stemp);

SR_FUNS( SET1:=Stemp,RESET:=Rtemp );
StartInterlock:=SR_FUNS.Q1;

(* Set  HornStartInterlock   Value  *)
HornStartInterlock:=StartInterlock
                                    AND (NOT EngineRun)
                                     AND MVL_POS_AHD_AST;

(* Set  HMI_StartInterlock   Value  *)
H_StartInterlock:=NOT ( FLASHER AND HornStartInterlock)
                                AND ( NOT EngineRun AND  StartInterlock);

(* Set  HMI_TurnGearEngaged   Value  *)
H_TurnGearEngaged:=NOT TurningGearDiseng;

(* Set  HMI_TurnGearSensorFail   Value  *)
H_TurnGearSensorFail:=TurningGearSensorFail;

(* Set  ShtLockDevEngaged  Value  *)
H_ShtLockDevEngaged:=ShaftLockingDeviceEngaged;

(*----------------------------------------------------------------*)
END_FUNCTION_BLOCK

(* POU ME_Start_Brake_Sequence, ST *)
FUNCTION_BLOCK ME_Start_Brake_Sequence
VAR_INPUT
END_VAR
VAR_OUTPUT
END_VAR
VAR
	TONInst: TON;(*TON()*)
	TONInst2: TON;(*TON()*)
       SRInst: SR; (*SR()*)
       SRInst2: SR; (*SR()*)

	tonQ: BOOL; (*store TOF.Q *)
       rsQ: BOOL; (*store  RS.Q1 / ENGINE RUN*)
	rs2Q: BOOL; (*store  RS.Q1 / ENGINE RUN*)


END_VAR
(*----------------4.1.5.2.2  ME Start, Break Sequence--------------*)

(*  set   BRAKE   Value   *)
BRAKE:=EngTurnINNonCRSPDir
        AND(NOT  NNBrake)
       AND( NOT(startFail OR startInterlock ));

(*  set   PRESTART   Value *)
TONInst(IN:=engineRun,PT :=RstartInhibitDelay);
 tonQ:=TONInst.Q;
 SRInst(SET1:=tonQ, RESET:=MVL_POS_STOP);
 rsQ:=SRInst.Q1;
SRInst2(SET1:=rsQ, RESET:=AllowRestartReset);
rs2Q:=SRInst2.Q1;

PRESTART:=NOT( startFail OR startInterlock)
                        AND (NOT rsQ)
	                 AND (MVL_POS_AHD OR MVL_POS_AST )
                        AND(EngineStandstill OR EngTurnINCRSPDir )
                        AND (NOT (NNstart  AND (NOT rs2Q)));

(*  set   START   Value   *)
START:= PRESTART
                AND  AnyAuxBlowerRun
                AND (  NOT SlowTurnRequestViaMVL);

(*  set   START,BREAK  BX7302C   Value   *)
START_BRAKE:=START  OR  BRAKE;

(*  set   ALLOWRESTARTRESET   Value   *)
TONInst2( IN:=START,  PT:= AllowRestartResetDelay );
AllowRestartReset:=TONInst2.Q;

(*  set   AHEAD   BX7302C  Value   *)
AHEAD:=MVL_POS_AHD AND RemoteCtrl ;

(*  set   ASTERN   BX7302C  Value   *)
ASTERN:=MVL_POS_AST AND RemoteCtrl;

(*  set   STOP   BX7302C  Value   *)
STOP:=NOT MVL_POS_AHD
              AND ( NOT MVL_POS_AST)
              AND RemoteCtrl;
END_FUNCTION_BLOCK

(* POU Slow_Turning_Sequence, ST *)
FUNCTION_BLOCK Slow_Turning_Sequence
VAR_INPUT
END_VAR
VAR_OUTPUT
END_VAR
VAR
	temp: BOOL;
	tonQ: BOOL;
	SR_FUNS: SR;

	temp1: BOOL;
	temp2: BOOL;


	TON_FUNS:TON;
	TON_FUNS2:TON;
	ecrautpbctrl: BOOL;
	brpushctrl: BOOL;


END_VAR
(*------------------4.1.5.2.3  SLOW TURNING SEQUENCE--------------------------*)

IF SLOWTURNOK OR ENGINERUN THEN POWERUP:=FALSE; END_IF;
(*---------------- Set SLOW  TURN.  REQUEST---------------- *)
temp:=SLOWTURNOK OR ENGINERUN;
TON_FUNS(IN:=(NOT temp),  PT:=SlowTurnDelayRequest);
tonQ:=TON_FUNS.Q;
SR_FUNS(SET1:=(tonQ OR POWERUP), RESET:=temp);
SlowTurnQuest:=SR_FUNS.Q1;


(*--------Set SLOW  TURN.  REQUEST. VIA    MVL------------*)
SlowTurnRequestViaMVL:=SlowTurnQuest AND  SlowByMVLEnable;

(*---------Set  HMI   SLOW  TURNING   Value-----------------*)
temp1:=(NOT SlowTurningBX) AND SlowTurnQuest;
(*temp2:=FLASHER_CTRL AND SlowTurningBX;*)(* TO HMI PULSE *)
temp2:= SlowTurningBX; (* TO HMI  NOT PULSE *)
H_SlowTurning:=temp1 OR temp2;

(*----------Set  SLOW  TURNFAILURE   Value---------------------------*)
SlowTurningFailure:=SlowTurnFailBX;

(*-----------Set  HMI  TURN FAIL RESET----------------*)
(*H_SlowTurnFailReset:=FLASHER_CTRL AND SlowTurnFailBX;*)(* TO HMI PULSE*)
H_SlowTurnFailReset:=  SlowTurnFailBX;(* TO HMI  NOT PULSE*)

(*-----------Set   SLOW TURN. RC  BX  Value ---------------------*)
temp:=MVL_POS_AHD OR MVL_POS_AST;

TON_FUNS2(IN:=temp, PT:=T#2s);
aheadastern:=TON_FUNS2.Q AND SlowTurnRequestViaMVL;
brpushctrl:=  SlowTurnBRPush AND BR_CTRL;
ecrautpbctrl:=SlowTurnECRAPush AND ECRA_CTRL;

SlowTurnRCBX:= (aheadastern OR brpushctrl OR ecrautpbctrl )
                                      AND  (NOT STARTINTERLOCK);


(*-------Set   SLOW TURN. FAIL RESET RC   BX  Value --------------   *)
SlowTurnFailResetRC:= (BR_CTRL AND  SlowTurnFailReset_BR_PU )
                                                       OR  ( ECRA_CTRL AND SlowTurnFailReset_ECRA_PU   );
END_FUNCTION_BLOCK

(* POU Air_Run_Sequence, ST *)
FUNCTION_BLOCK Air_Run_Sequence
VAR_INPUT
END_VAR
VAR_OUTPUT
END_VAR
VAR
	AIRRUN_RC_BX: BOOL;
END_VAR
(*----------4.1.5.2.4 Air Run Sequence------------------------*)
AIRRUN_RC_BX:= (AIRRUN AND ECRA_CTRL)
                                          AND(NOT  STARTINTERLOCK)
                                          AND ( EngineStandstill OR  AIRRUN_RC_BX);

H_AIRRUN_BR_ECR:=AIRRUN_RC_BX;
END_FUNCTION_BLOCK

(* POU Auxiliary_Blower, ST *)
FUNCTION_BLOCK Auxiliary_Blower
VAR_INPUT
END_VAR
VAR_OUTPUT
END_VAR
VAR
	SR_FUNS: SR;
END_VAR
(*-----------------4.1.5.2.5 AUXILIARY BLOWER-----------------*)

(*SET HMI AUTO.BLOWER.MAN.CONTROL *)
H_AuxBlowerManCTRL:=AuxBlowerManCTRL;

AuxBlower_preslct_rc_ready:=(AuxBlowerReselECRA_PB AND ECRA_CTRL AND  NOT SAFETY_SYSTEM_OFF_FAIL);
SR_FUNS(SET1:=AuxBlower_preslct_rc_ready,RESET:=AuxBlowerStop_PB  AND  ECRA_CTRL );

(*SET AUX_BLOWER_PRESELECTED_RC *)
AuxBlowerPreselectedRC:=SR_FUNS.Q1;

(*SET HMI_AUX_BLOWER_PRESEL *)
H_AuxBlowerPresel:=SR_FUNS.Q1;

(* Set AUX.BLOWER FAILED  Value*)
H_AuxBlowerFailed:=AuxBlowerFailed;
(*-------------------------------------------------------------------------------------*)
END_FUNCTION_BLOCK

(* POU Crank_Angle_System, ST *)
FUNCTION_BLOCK Crank_Angle_System
VAR_INPUT
END_VAR
VAR_OUTPUT
END_VAR
VAR

END_VAR
(*---------4.1.5.2.6 CRANK ANGLE SYSTEM----------------- *)

(* STARTLEARNINGINPROGRESSstatus:=STARTLEARNINGINPROGRESS;AND FLASHER?????????????*)

H_StartLearningInPro:=StartLearningInPro;(* AND FLASHER?????????????*)
(*---------------------------------------------- *)
END_FUNCTION_BLOCK

(* POU Control_Transfer, ST *)
FUNCTION_BLOCK Control_Transfer
VAR_INPUT
END_VAR
VAR_OUTPUT
END_VAR
VAR

END_VAR
(*-----------------4.1.5.2.7 CTRL  TRANSFER  ------------  *)

RemoteCtrl:= BR_CTRL OR ECRA_CTRL;

(*--------------------------CONTROL    TRANSFER---------------------------*)
(*----------------------------------------------------------INPUT-------------------------------------------------------------------*)
(*-----------------------------BR------------------------------*)(*Page 29.04*)
       BR_PUS_SGNL_BR_CTRL:=BR_PUS_BR_CTRL;
	BR_PUS_SGNL_ECRA_CTRL:=BR_PUS_ECRA_CTRL;
	BR_PUS_SGNL_ECRM_CTRL:=BR_PUS_ECRM_CTRL;
	BR_PUS_SGNL_LOC_MAN_CTRL:=BR_PUS_LOC_MAN_CTRL;

(*------------------------------ECR-------------------------------*)
	ECRA_PUS_SGNL_BR_CTRL:=ECRA_PUS_BR_CTRL;
	ECRA_PUS_SGNL_ECRA_CTRL:=ECRA_PUS_ECRA_CTRL;
	ECRA_PUS_SGNL_ECRM_CTRL:=ECRA_PUS_ECRM_CTRL;
	ECRA_PUS_SGNL_LOC_MAN_CTRL:=ECRA_PUS_LOC_MAN_CTRL;

(*------------------------------------------------------------------OUTPUT----------------------------------------------------------*)

(*------------------------BR-------------------------*)
      BR_LAMPS_BR_CTRL:=  (BRG_BRG_CTRL_FLSH AND  FLASHER)
                                                         OR  ( ( NOT BRG_BRG_CTRL_FLSH) AND BR_CTRL ) ;


      BR_LAMPS_ECRA_CTRL:= (BRG_ECRA_CTRL_FLSH AND FLASHER)
                                                             OR   ((NOT BRG_ECRA_CTRL_FLSH)  AND ECRA_CTRL);

      BR_LAMPS_ECRM_CTRL:=(BRG_ECRM_CTRL_FLSH AND FLASHER)
                                                             OR   ((NOT BRG_ECRM_CTRL_FLSH)  AND  ECRM_CTRL);

      BR_LAMPS_LOCAL_MAN_CTRL:=(BRG_LOCAL_MAN_CTRL_FLSH AND FLASHER)
                                                                      OR ((NOT BRG_LOCAL_MAN_CTRL_FLSH ) AND  LOC_MAN_CTRL);

      BR_ACCOUST_SIGN_CTRL:=BR_ACCOUST_CTRL_SIGN_BX;

       H_HORN_ALARM_BRG:=BR_ACCOUST_SIGN_CTRL;(*HMI  ALARM SPEAKER*)

(*----------PORT/ STBD TO CONTRL THE BR_IN_CTRL light ON/OFF-------------*)
      IF ((PORT_CTRL_EOT OR STBD_CTRL_EOT) AND BR_CTRL)
      THEN
         BR_BRIDGE_IN_CONTROL:= FALSE;
         BR_LAMPS_BR_CTRL:=FALSE;
      END_IF
(*--------PORT/ STBD TO CONTRL THE BR_IN_CTRL light ON/OFF-----------*)


(*-----------------------ECR-------------------------*)
     ECR_LAMPS_BR_CTRL:=  (ECR_BRG_CTRL_FLSH AND  FLASHER)
                                                          OR  ( ( NOT ECR_BRG_CTRL_FLSH) AND BR_CTRL ) ;

      ECR_LAMPS_ECRA_CTRL:= (ECR_ECRA_CTRL_FLSH AND FLASHER)
                                                              OR   ((NOT ECR_ECRA_CTRL_FLSH)  AND ECRA_CTRL);

      ECR_LAMPS_ECRM_CTRL:=(ECR_ECRM_CTRL_FLSH AND FLASHER)(* ------------没有硬线地址------------*)
                                                               OR   ((NOT ECR_ECRM_CTRL_FLSH)  AND  ECRM_CTRL);

     ECR_LAMPS_LOCAL_MAN_CTRL:=(ECR_LOCAL_MAN_CTRL_FLSH AND FLASHER)
                                                                          OR ((NOT ECR_LOCAL_MAN_CTRL_FLSH ) AND  LOC_MAN_CTRL);

     ECR_ACCOUST_SIGN_CTRL:=ECR_ACCOUST_CTRL_SIGN_BX;

     H_HORN_ALARM_ECR:=ECR_ACCOUST_SIGN_CTRL;(*HMI ALARM SPEAKER*)
END_FUNCTION_BLOCK

(* POU Speed_Control, ST *)
FUNCTION_BLOCK Speed_Control
VAR_INPUT
END_VAR
VAR_OUTPUT
END_VAR
VAR
	BR_SEARCH_COUNTER_INST:  SearchRPM_By_ELEC;
       BR_LEVEL_INST:CAL_K_B;

	ECR_SEARCH_COUNTER_INST:  SearchRPM_By_ELEC;
       ECR_LEVEL_INST:CAL_K_B;

	FREEZE: BOOL;
	TONInst:TON;
	TONQ: BOOL;
	LIMIT_TEMP: REAL;(*LIMIT temp value *)
	TEMPVALUE: REAL;
	SEARCHRPMInst:  SearchRPM_By_ELEC;
	SEARCHRPMInst_wgf:  SearchRPM_By_ELEC;
	SEARCHRPMInst_wgf124:  SearchRPM_By_ELEC;
      CAL_K_BInst:CAL_K_B;
	CAL_K_BInst_wgf:CAL_K_B;
	CAL_K_BInst_wgf124:CAL_K_B;
	RAMP_REALInst:RAMP_REAL;
	DIFFER: REAL;
	Temp_Time: TIME;
	Rate_Change: REAL;
	OVER_SPEED_TEMP: BOOL;
	SRInst: SR;

	RTRIG_INST: R_TRIG;

	TEMPQ: BOOL;
	FREEZE_SR: SR;

	FLAG_STOP: BOOL;
	MVL_FINE_ADJUST_INCREASE:BOOL;
	MVL_FINE_ADJUST_DECREASE:BOOL;
	MVL_FINE_ADJUST_START_TEMP:BOOL;
	MVL_FINE_ADJUST_START_RISE:BOOL;
	SRStart_fine_adjust:SR;
	R_TRIG_FINE_incr:R_TRIG;
	R_TRIG_FINE_decr:R_TRIG;
	R_TRIG_FINE_START:R_TRIG;
	CONT_MVL_CMD_FINE_START:REAL;

END_VAR
(* -----------------WRONG_WAY-----------------*)
IF(    (ECRM_CTRL OR  LOC_MAN_CTRL) AND  EngTurnINNonCRSPDir)
THEN
WRONG_WAY_ALARM:=TRUE;
ELSE
WRONG_WAY_ALARM:=FALSE;
END_IF;


(*-----------------PROPULSION CONTROL PASSIVE  FAILURES------------------------------  *)
propulsion_ctrl_passive_failure_alm:=MVL_BR_FAIL OR MVL_ECR_FAIL
                                                                       OR RCS_SPD_SENSOR_FAIL1 OR RCS_SPD_SENSOR_FAIL2 ;

(*------------------PROPULSION CONTROL FAILURES--------------------------------*)
propulsion_ctrl_failure_alm:=MVL_BR_FAIL OR MVL_ECR_FAIL  OR PCS_POWER_SUPPLY_ALM;
Propulsion_Control_Failure_ALM:= NOT propulsion_ctrl_failure_alm;


(* ---------------------------4.1.5.2.8 SPEED MEASURE---------------------------------*)
IF ( RCS_SPD_SENSOR_FAIL1 OR RCS_SPD_SENSOR_FAIL2)
THEN
 PCS_SPD_MEASURE_FAILURE:=TRUE;
ELSE
PCS_SPD_MEASURE_FAILURE:=FALSE;
END_IF

SRInst(SET1:=OVERSPEED_RCS_TEMP , RESET:=((NOT OVERSPEED_RCS_TEMP)   AND   MVL_POS_STOP));
RCS_SW_overspd:= SRInst.Q1;

OVER_SPEED:=RCS_SW_overspd OR RCS_HW_overspd;

 eng_tripped:=OVER_SPEED OR SafetyStop;


(* calculate the position of the EOT( BR and ECR) and the value will dispaly to  the HMI*)
(*EOT LEVEL OF BR  *)
(*
BR_SEARCH_COUNTER_INST(ELEC_SEARCH:=MVL_POSITION_BR);
BR_LEVEL_INST(counter:=BR_SEARCH_COUNTER_INST.Counter, ECE_VALUE:=MVL_POSITION_BR);
BR_MVL_LEVEL:=BR_LEVEL_INST.POSITION;

(*EOT LEVEL OF ECR  *)
ECR_SEARCH_COUNTER_INST(ELEC_SEARCH:= MVL_POSITION_ECR );
ECR_LEVEL_INST(counter:=ECR_SEARCH_COUNTER_INST.Counter, ECE_VALUE:=MVL_POSITION_ECR);
ECR_MVL_LEVEL:=ECR_LEVEL_INST.POSITION;
*)

(* ---------------------4.1.5.2.9 Speed Control---------------------*)
(*EOT LEVEL OF BR  *)
BR_SEARCH_COUNTER_INST(ELEC_SEARCH:=MVL_POSITION_BR  );
BR_LEVEL_INST(counter:=BR_SEARCH_COUNTER_INST.Counter, ECE_VALUE:=MVL_POSITION_BR);
BR_MVL_LEVEL:=BR_LEVEL_INST.POSITION;

(*EOT LEVEL OF ECR  *)
ECR_SEARCH_COUNTER_INST(ELEC_SEARCH:= MVL_POSITION_ECR );
ECR_LEVEL_INST(counter:=ECR_SEARCH_COUNTER_INST.Counter, ECE_VALUE:=MVL_POSITION_ECR);
ECR_MVL_LEVEL:=ECR_LEVEL_INST.POSITION;
(*-------SET  MVL_BR_FAIL  VALUE-------------*)
IF(NOT (MVL_POSITION_BR >MVL_FAIL_VALUE))
THEN    MVL_BR_FAIL:=TRUE;
ELSE    MVL_BR_FAIL:=FALSE;
END_IF;

(*--------SET  MVL_FAILURE  VALUE-----------*)
MVL_FAILURE:=(MVL_BR_FAIL AND BR_CTRL)
                             OR (MVL_ECR_FAIL AND ECRA_CTRL) ;

(*--------SET  MVL_ECR_FAIL   VALUE---------*)
IF(NOT (MVL_POSITION_ECR >MVL_FAIL_VALUE))
THEN   MVL_ECR_FAIL:=TRUE;
ELSE   MVL_ECR_FAIL:=FALSE;
END_IF;

(* SPEED_SET_SIGNALA*)
(*----------FREEZE----------------*)
RTRIG_INST(CLK:=MVL_POS_STOP);
IF RTRIG_INST.Q
THEN
      	FREEZE := TRUE;
       FLAG_STOP:=TRUE;
END_IF

IF FLAG_STOP
THEN
     TONInst( IN:= TRUE,  PT:=PULSE_TIME);
END_IF

 IF TONInst.Q
THEN
      	FREEZE := FALSE;
      TONInst( IN:= FALSE,  PT:=PULSE_TIME);
       FLAG_STOP:=FALSE;
END_IF


(*(*Set FREEZE Value      once EOT leave  the stop place,the  FREEZE is set  to FALSE. *)
IF ( BR_CTRL  AND  ( MVL_POSITION_BR>MVL_POS_AHEAD_VALUE  OR   MVL_POSITION_BR< MVL_POS_ASTERN_VALUE ))(* this means  that BR  EOT is not  stop  place *)
THEN
   FREEZE:=FALSE;
END_IF;
IF (ECRA_CTRL AND  (MVL_POSITION_ECR>MVL_POS_AHEAD_VALUE OR   MVL_POSITION_ECR< MVL_POS_ASTERN_VALUE ))
THEN
   FREEZE:=FALSE;
END_IF;*)
(*--------------------------*)

IF( NOT  FREEZE)THEN
       (*select  change rate and  save rate in  Rate_Change *)
      IF(SHAFT_GENERATOR_BREAKER)
      THEN
             Rate_Change:=RATE_OF_CHANGE_SLOW;
      ELSE
             Rate_Change:=RATE_OF_CHANGE_FAST;
      END_IF;
             Rate_Change:=ConvertValue*Rate_Change;

         (*select control right  (BR OR ECTA)  and save target  elec in  Target_Elec *)
  (*    IF(BR_CTRL)(*when control right in BR*)
           THEN    Target_Elec:=MVL_POSITION_BR;
      ELSIF(ECRA_CTRL)  (*when control right in ECR AUTO*)
           THEN    Target_Elec:=MVL_POSITION_ECR;
      ELSE
             Target_Elec:=MVL_STOP_VALUE;
      END_IF;*)
	   IF(BR_CTRL)(*when control right in BR*)
           THEN    Target_Elec:=MVL_POSITION_BR;
      ELSE
             Target_Elec:=MVL_POSITION_ECR;
      END_IF;
      (* RAMP function*)
     		RAMP_REALInst(IN:=Target_Elec, ASCEND:=Rate_Change*0.01,DESCEND:=Rate_Change*0.01, TIMEBASE:=T#0.01s,RESET:=FALSE);
    		 SPEED_SET_SIGNALA:=RAMP_REALInst.OUT;
ELSE(* IF  FREEZE , Target_Elec will equal to current value*)
     RAMP_REALInst(IN:=RAMP_REALInst.OUT, ASCEND:=Rate_Change*0.01, DESCEND:=Rate_Change*0.01, TIMEBASE:=T#0.01s,RESET:=FALSE);
     SPEED_SET_SIGNALA:=RAMP_REALInst.OUT;
  END_IF;
(*--------Set   MVLAHEAD  Value-------- *)
IF(SPEED_SET_SIGNALA>MVL_POS_AHEAD_VALUE)
THEN MVL_POS_AHD:=TRUE;
ELSE MVL_POS_AHD:=FALSE;
END_IF;

(*--------Set   MVLASTERN  Value --------*)
IF(NOT(SPEED_SET_SIGNALA>MVL_POS_ASTERN_VALUE))
THEN MVL_POS_AST:=TRUE;
ELSE MVL_POS_AST:=FALSE;
END_IF;

(*--------Set   MVL_POS_AHD_AST  Value-------- *)
 MVL_POS_AHD_AST:=MVL_POS_AHD OR MVL_POS_AST;

(*--------Set   MVLSTOP  Value-------- *)
 MVL_POS_STOP:=NOT MVL_POS_AHD_AST;




(*-------------------------------------------------------MVLFINE FUNCTION---------------------------------------------------------------------------------------------*)
																			(*----------Get the CMD from HMI-------------*)
	IF h_speed_cmd_adjust_mb=1 THEN
	MVL_FINE_ADJUST_INCREASE:=TRUE;
	ELSE
	MVL_FINE_ADJUST_INCREASE:=FALSE;
	END_IF

	IF h_speed_cmd_adjust_mb=-1 THEN
	MVL_FINE_ADJUST_DECREASE:=TRUE;
	ELSE
	MVL_FINE_ADJUST_DECREASE:=FALSE;
	END_IF              (*解析HMI发下来的命令，加速or减速*)
	R_TRIG_FINE_incr(CLK:=MVL_FINE_ADJUST_INCREASE);
	MVL_FINE_ADJUST_INCREASE_RISE:=R_TRIG_FINE_incr.Q;(*加速按钮上升沿信号*)
	R_TRIG_FINE_decr(CLK:=MVL_FINE_ADJUST_DECREASE);
	MVL_FINE_ADJUST_DECREASE_RISE:=R_TRIG_FINE_decr.Q;(*减速按钮上升沿信号*)
																			(*----------Start fine adjust function  (available)-------------*)
	IF RemoteCtrl AND  h_speed_cmd_adjust_mb<>0 AND  EngineRun THEN
	MVL_FINE_ADJUST_START_TEMP:=TRUE;
	ELSE
	MVL_FINE_ADJUST_START_TEMP:=FALSE;
	END_IF
	SRStart_fine_adjust(SET1:=MVL_FINE_ADJUST_START_TEMP,RESET:=MVL_MOVE OR (NOT RemoteCtrl));(*若车钟移动则退出*)
	MVL_FINE_ADJUST_AVAILABLE:=SRStart_fine_adjust.Q1;
	R_TRIG_FINE_START(CLK:=MVL_FINE_ADJUST_AVAILABLE);
	MVL_FINE_ADJUST_START_RISE:=R_TRIG_FINE_START.Q;(*检测进入微调状态上升沿*)
																			(*----------Detect MVL moved during fine adjustnig-------------*)
	IF	MVL_FINE_ADJUST_START_RISE THEN
		IF BR_CTRL THEN CONT_MVL_CMD_FINE_START:=BR_MVL_RPM_CMD; END_IF
		IF ECRA_CTRL THEN CONT_MVL_CMD_FINE_START:=MCR_MVL_RPM_CMD; END_IF
	END_IF  (*进入微调状态采样*)

	IF MVL_FINE_ADJUST_AVAILABLE THEN
	 	IF BR_CTRL AND ((BR_MVL_RPM_CMD-CONT_MVL_CMD_FINE_START>SPT_mvl_fine_reset) OR  (CONT_MVL_CMD_FINE_START-BR_MVL_RPM_CMD>SPT_mvl_fine_reset))THEN MVL_MOVE:=TRUE; END_IF
		IF ECRA_CTRL AND ((MCR_MVL_RPM_CMD-CONT_MVL_CMD_FINE_START>SPT_mvl_fine_reset) OR (CONT_MVL_CMD_FINE_START-MCR_MVL_RPM_CMD>SPT_mvl_fine_reset)) THEN MVL_MOVE:=TRUE; END_IF(*判断车钟是否动作*)
	ELSE
		MVL_MOVE:=FALSE;
	END_IF

																			(*----------Fine Adjust Value-------------*)
	IF MVL_FINE_ADJUST_AVAILABLE THEN
		IF MVL_FINE_ADJUST_INCREASE_RISE THEN FINE_ADJUST_VALUE:=FINE_ADJUST_VALUE+SPT_mvl_fine_stage; END_IF
		IF MVL_FINE_ADJUST_DECREASE_RISE THEN FINE_ADJUST_VALUE:=FINE_ADJUST_VALUE-SPT_mvl_fine_stage; END_IF
	ELSE
		FINE_ADJUST_VALUE:=0;
	END_IF



(*--------------SET SPEED_SET_SIGNALB  VALUE;--------------------------------------------------------------------------------------------------------------------------------------*)

IF  SPEED_SET_SIGNALA>MVL_POS_ASTERN_VALUE AND SPEED_SET_SIGNALA<MVL_POS_AHEAD_VALUE(* IF target  Elec value between 11mA and 12mA , SPEED_SET_SIGNALB=0*)(*MVL_POS_AHEAD_VALUE=13mA   MVL_POS_ASTERN_VALUE=11mA  POS.=STOP*)
	 THEN  SPEED_SET_SIGNALB:=0;
ELSIF  SPD_SIM_MODE_ACTIVE<0.5(*如果当前为仿真模式，将仿真得到的RCS_SPEED_MEANSURE_VALUE反馈给 SPEED_SET_SIGNALB -----  AND    SMI_SPD_FROM_HMI>0.5   TARGET_VALUE: 1:target from HMI   0:target  from MVL *)
      THEN  SPEED_SET_SIGNALB:= RCS_SPEED_MEANSURE_VALUE;
ELSE (*如果不是上述两种情况的话，其逻辑按照图上进行处理*)
SEARCHRPMInst(ELEC_SEARCH:= SPEED_SET_SIGNALA );
CAL_K_BInst(counter:=SEARCHRPMInst.Counter, ECE_VALUE:=SPEED_SET_SIGNALA);
SPEED_SET_SIGNALB:=SPEED_SET_SIGNALA*CAL_K_BInst.K_VALUE+CAL_K_BInst.B_VALUE +FINE_ADJUST_VALUE;
END_IF;


(*-----------------SET SPEED_SET_SIGNALC VALUE----------------------*)
IF( SLOW_DOWN )
      THEN
       IF (SLOW_DOWN_VALUE<SPEED_SET_SIGNALB)  THEN  SPEED_SET_SIGNALC:=SLOW_DOWN_VALUE;
        ELSE SPEED_SET_SIGNALC:=SPEED_SET_SIGNALB;
        END_IF;
ELSE
     SPEED_SET_SIGNALC:=SPEED_SET_SIGNALB;
END_IF;


(* SET  SPEED_SETPOINT_BX VALUE*)
LIMIT_TEMP:=LIMIT(LO_CHIEF_LIMIT,CHIEFLIMIT, MAX_SPEED);
IF(LIMIT_TEMP<SPEED_SET_SIGNALC)
THEN SPEED_SETPOINT_BX:=LIMIT_TEMP;
ELSE SPEED_SETPOINT_BX:=SPEED_SET_SIGNALC;
END_IF;

(*Set HMI_ BR&ECR MVL_RPM_CMD  Value*)
					(*BR*)
	IF  MVL_POSITION_BR>MVL_POS_ASTERN_VALUE AND MVL_POSITION_BR<MVL_POS_AHEAD_VALUE(* IF mvl position value between 11mA and 12mA , SPEED_SET_SIGNALB=0*)(*MVL_POS_AHEAD_VALUE=13mA   MVL_POS_ASTERN_VALUE=11mA  POS.=STOP*)
      THEN  BR_MVL_RPM_CMD:=0;
	ELSE
	SEARCHRPMInst_wgf(ELEC_SEARCH:= MVL_POSITION_BR );
	CAL_K_BInst_wgf(counter:=SEARCHRPMInst_wgf.Counter, ECE_VALUE:=MVL_POSITION_BR);
	BR_MVL_RPM_CMD:=MVL_POSITION_BR*CAL_K_BInst_wgf.K_VALUE+CAL_K_BInst_wgf.B_VALUE;
	END_IF;
					(*MCR*)
	IF  MVL_POSITION_ECR>MVL_POS_ASTERN_VALUE AND MVL_POSITION_ECR<MVL_POS_AHEAD_VALUE(* IF mvl position value between 11mA and 12mA , SPEED_SET_SIGNALB=0*)(*MVL_POS_AHEAD_VALUE=13mA   MVL_POS_ASTERN_VALUE=11mA  POS.=STOP*)
      THEN  MCR_MVL_RPM_CMD:=0;
	ELSE
	SEARCHRPMInst_wgf124(ELEC_SEARCH:= MVL_POSITION_ECR );
	CAL_K_BInst_wgf124(counter:=SEARCHRPMInst_wgf124.Counter, ECE_VALUE:=MVL_POSITION_ECR);
	MCR_MVL_RPM_CMD:=MVL_POSITION_ECR*CAL_K_BInst_wgf124.K_VALUE+CAL_K_BInst_wgf124.B_VALUE;
	END_IF;
(*Set   HMI_BR_ECRA_CHIEFLIMIT  Value*)
IF(SPEED_SET_SIGNALC -  LIMIT_TEMP>0)
THEN  HMI_BR_ECRA_CHIEFLIMIT:=TRUE;
ELSE  HMI_BR_ECRA_CHIEFLIMIT:=FALSE;
END_IF;

(* Set   RC_HANDLE_MATCH  Value *)
TEMPVALUE:=ABS(MVL_POSITION_BR-MVL_POSITION_ECR);
IF(NOT(TEMPVALUE>MVL_HANDLE_MATCH))
       THEN    RC_HANDLE_MATCH:=TRUE;
ELSE RC_HANDLE_MATCH:=FALSE;
END_IF;
(* Send   RC_HANDLE_MATCH  to HMI *)
H_MVL_HANDLE_MATCH_mb:=RC_HANDLE_MATCH;

(*-----------------SET SPEED_SET_SIGNALC VALUE----------------------*)
(*IF(LOAD_LIMIT_IN_GAS_MODE)
THEN
        IF(LOAD_LIMIT_IN_GAS_MODE_VALUE<SPEED_SET_SIGNALB)  THEN  SPEED_SET_SIGNALC:=LOAD_LIMIT_IN_GAS_MODE_VALUE;(*?????????????*)
        ELSE SPEED_SET_SIGNALC:=SPEED_SET_SIGNALB;
        END_IF;
IF( SLOW_DOWN )
THEN
        IF(SLOW_DOWN_VALUE<SPEED_SET_SIGNALB)  THEN  SPEED_SET_SIGNALC:=SLOW_DOWN_VALUE;
        ELSE SPEED_SET_SIGNALC:=SPEED_SET_SIGNALB;
        END_IF;
ELSE
        IF(MAX_VALUE<SPEED_SET_SIGNALB)  THEN  SPEED_SET_SIGNALC:=MAX_VALUE;
        ELSE SPEED_SET_SIGNALC:=SPEED_SET_SIGNALB;
        END_IF;
END_IF;*)

(* *)
END_FUNCTION_BLOCK

(* POU SearchRPM_By_ELEC, ST *)
FUNCTION_BLOCK SearchRPM_By_ELEC
VAR_INPUT
	ELEC_SEARCH: REAL;
END_VAR
VAR_OUTPUT
	Counter: INT;
END_VAR
VAR
	FLAG: BOOL;
	RPM_VALUE: REAL;
	RATE: REAL;

END_VAR
IF(ELEC_SEARCH<=GRADE_RPM_ELEC_MAP[5].ELEC)THEN
       FOR Counter:=6 TO 10 BY 1 DO
            IF(ELEC_SEARCH>=GRADE_RPM_ELEC_MAP[Counter].ELEC)THEN
                   RPM_VALUE:=GRADE_RPM_ELEC_MAP[Counter].RPM;
                   RPM_VALUE:=GRADE_RPM_ELEC_MAP[Counter].GRADE;
                   EXIT;
            END_IF;
      END_FOR;
ELSE
    FOR Counter:=4 TO 0  BY -1 DO
            IF(ELEC_SEARCH<=GRADE_RPM_ELEC_MAP[Counter].ELEC)THEN
                   RPM_VALUE:=GRADE_RPM_ELEC_MAP[Counter].RPM;
                   RPM_VALUE:=GRADE_RPM_ELEC_MAP[Counter].GRADE;
                   EXIT;
            END_IF;
      END_FOR;
END_IF;
END_FUNCTION_BLOCK

(* POU CAL_K_B, ST *)
FUNCTION_BLOCK CAL_K_B
VAR_INPUT
	counter: INT;
       ECE_VALUE:REAL;

END_VAR
VAR_OUTPUT
	K_VALUE: REAL;
	B_VALUE: REAL;
	POSITION: REAL;(* 档位*)

END_VAR
VAR
	POS: INT;
	value1: REAL;
	value2: REAL;

END_VAR
IF(GRADE_RPM_ELEC_MAP[counter].ELEC<=GRADE_RPM_ELEC_MAP[5].ELEC)THEN
pos:=counter-1;
ELSE
POS:=counter;
END_IF;

value1:=(GRADE_RPM_ELEC_MAP[pos+1].RPM-GRADE_RPM_ELEC_MAP[pos].RPM);
value2:=(GRADE_RPM_ELEC_MAP[pos+1].ELEC -GRADE_RPM_ELEC_MAP[pos].ELEC);

K_VALUE:=value1/value2;

B_VALUE:=GRADE_RPM_ELEC_MAP[pos].RPM   -   K_VALUE*GRADE_RPM_ELEC_MAP[pos].ELEC;


POSITION:=POS+ABS(ECE_VALUE-GRADE_RPM_ELEC_MAP[pos].ELEC) / ABS(value2);
END_FUNCTION_BLOCK

(* POU Crash_Reverse, ST *)
FUNCTION_BLOCK Crash_Reverse
VAR_INPUT
END_VAR
VAR_OUTPUT
END_VAR
VAR
	TOFInst:TOF;
	FLAG: BOOL;
	B_Value: REAL;
	K_VaLue: REAL;
END_VAR
(*--------------------4.1.5.2.10 Crash Reverse-----------------------*)


       (*reset the  timer*)
       TOFInst(IN:= TRUE, PT:= T#1ms);
       TOFInst.Q;
(*

K_Value:=200.0/(GRADE_RPM_ELEC_MAP[0].ELEC-GRADE_RPM_ELEC_MAP[10].ELEC);
B_Value:= 100.0-GRADE_RPM_ELEC_MAP[0].ELEC*K_Value;
EOT_LEVER_VAULE:=REAL_TO_INT(Target_Elec*K_Value+B_Value);

(*check current lever value  above the up limit*)
IF( EOT_LEVER_VAULE >= Enable_Crash_Astern_S1)
THEN
	CA_ABOVE_LIMIT_FLAG := TRUE;
END_IF

(*when the lever value change from upper 90 to lower 90*)
IF (CA_ABOVE_LIMIT_FLAG AND EOT_LEVER_VAULE < Enable_Crash_Astern_S1 )
THEN
	(*start timer,2S delay*)
	TOFInst(IN:= FALSE, PT:=CrashMovDly);
	CA_ABOVE_LIMIT_FLAG := FALSE;
       FLAG:=TRUE;
END_IF

(*wait until timer  counts end*)
IF (TOFInst.Q AND  FLAG)
THEN
	(*if the lever value less than -85,then active the CRASH ASTER MODE*)
	IF	(EOT_LEVER_VAULE <=Activate_Crash_Astern_S2)  (*  EOT CURRENT  POSITION*)
	THEN
		REVERSE_ACTIVE_SIGNAL := TRUE;
             FLAG:=FALSE;
      ELSE
             REVERSE_ACTIVE_SIGNAL := FALSE;
	END_IF
END_IF
(* CRASH ASTER MODE*)
IF	( REVERSE_ACTIVE_SIGNAL )
THEN
     CRASH_REVERSE_SPEEDPROGRAMOVERRIDE:=TRUE;
     CRASH_REVERSE_CANCELL_LIMITS:=TRUE;

(* exit the CRASH ASTER MODE*)

IF (( EngTurningAST AND  RCS_SPEED_MEANSURE_VALUE >ABS( REAL_Crash_Astern_S3)) OR  EOT_LEVER_VAULE  >Activate_Crash_Astern_S2)
	THEN
		REVERSE_ACTIVE_SIGNAL := FALSE;
	      CRASH_REVERSE_SPEEDPROGRAMOVERRIDE:=FALSE;
             CRASH_REVERSE_CANCELL_LIMITS:=FALSE;
	END_IF

END_IF

-----------------------------------------------------------------------------------------------------------------------------------------do not useing this funtionnal----------*)
END_FUNCTION_BLOCK

(* POU Simulation_Mode, ST *)
FUNCTION_BLOCK Simulation_Mode
VAR_INPUT
END_VAR
VAR_OUTPUT
END_VAR
VAR

	EOT_POS: INT;
	FLAG: BOOL;

END_VAR
(*------------------------4.1.5.2.11   ---------------------*)

IF(SPD_SIM_MODE_ACTIVE<0.5)(* 1:SHIP  0:TESBED*)
THEN
     SPD_SIM_MODE_ACTIVE_FLAG:=TRUE;
     IF(SMI_SPD_FROM_HMI>0.5)(*TARGET_VALUE: 1:HMI   0:MVL*)
     THEN
	      SIMULATION_TARGET_VALUE:=SIMULATION_TARGET_VALUE_FROMHMI;
      ELSE
	      SIMULATION_TARGET_VALUE:=SPEED_SETPOINT_BX ;
      END_IF;
ELSE
SPD_SIM_MODE_ACTIVE_FLAG:=FALSE;
END_IF
END_FUNCTION_BLOCK

(* POU Other_Function, ST *)
FUNCTION_BLOCK Other_Function
VAR_INPUT
END_VAR
VAR_OUTPUT
END_VAR
VAR
	TONInst:TON;
	HYSTERESISInst :HYSTERESIS;
	HYSTERESISInst2 :HYSTERESIS;
       RAMP_SPDTESTInst:RAMP_REAL;

	SpeedValue: INT;
	HIGHValue: INT;
	LOWValue: INT;
	BreakHValue: INT;
	BreakLValue: INT;


END_VAR
(* ------------------------P16.07------------------------------------------*)
(* -----------------------SPEED THRESHOLDS----------------------*)
  (*set   NNSTART*)
SpeedValue:=REAL_TO_INT(RCS_SPEED_MEANSURE_VALUE);(*SPEED MEAS. VALUE*)
HIGHValue:=REAL_TO_INT( NStartHIGH);(*NStartHIGH*)
LOWValue:=REAL_TO_INT(NStartLOW);(*NStartLOW*)
HYSTERESISInst(IN:=SpeedValue,  HIGH:=HIGHValue,   LOW:=LOWValue);
NNSTART:= NOT HYSTERESISInst.OUT;

(* SET NNBRAKE  *)
BreakHValue:=REAL_TO_INT(NBreakHIGH);(*NBreakHIGH*)
BreakLValue:=REAL_TO_INT(NBreakLOW);(*NBreakLOW*)
HYSTERESISInst(IN:=SpeedValue, HIGH:=BreakHValue,   LOW:=BreakLValue);
NNBRAKE:=NOT HYSTERESISInst.OUT;


(* -----------------ENG. TURNING IN  CORRESPONDING  NON-CORRESPONDING  DIRECTION-----------------*)
EngTurnINCRSPDir:= (MVL_POS_AHD AND EngTurningAHD)
                               OR ( MVL_POS_AST AND EngTurningAST  );

EngTurnINNonCRSPDir:=(MVL_POS_AHD AND  EngTurningAST)
                                           OR(EngTurningAHD AND  MVL_POS_AST );

(*------------------------ENGINE  RUNNING ------------------------*)
TONInst(IN:=(  EngTurnINCRSPDIR AND NNSTART),    PT:=EngineRuningDelay);
EngineRun:=TONInst.Q;

(*--------------------START AIR PRESSURE-------------------------*)
StartAirPress:=StartAirPressBX;(*0-4000 bar*)
HYSTERESISInst2( IN:=REAL_TO_INT(StartAirPress), HIGH:=REAL_TO_INT(StartAirPreHIGH*100),   LOW:=REAL_TO_INT(StartAirPreLOW*100));
StartAirPressLow:=HYSTERESISInst2.OUT;
H_StartAirPressLow:=HYSTERESISInst2.OUT;
(*
StartAirPress:=StartAirPressBX/100;(*0-4000~0-40*)
HYSTERESISInst2( IN:=REAL_TO_INT(StartAirPress), HIGH:=REAL_TO_INT(StartAirPreHIGH),   LOW:=REAL_TO_INT(StartAirPreLOW));
StartAirPressLow:=HYSTERESISInst2.OUT;
H_StartAirPressLow:=HYSTERESISInst2.OUT;
*)

(*------------------------START   FAILURE-------------------------------------------------------*)

startFail:=Start_Failure_BX;
(*Start_Fail_Flash_sign:=Start_Failure_BX AND  FLASHER_CTRL ;*)(* TO HMI PULSE *)
Start_Fail_Flash_sign:=Start_Failure_BX  ;(* TO HMI NOT PULSE *)
END_FUNCTION_BLOCK

(* POU Me_Over_Limit, ST *)
FUNCTION_BLOCK Me_Over_Limit
VAR_INPUT
END_VAR
VAR_OUTPUT
END_VAR
VAR






END_VAR
(*------------------NO16-ME OVER LIMIT------------------------------*)

(* SPEED OVERRIDE     *)
SPEED_PRGM_OVERD_BX:= ( SPEED_PRGM_OVERRIDE_BR AND BR_CTRL)
                                                     OR  (  SPEED_PRGM_OVERRIDE_ECA  AND ECRA_CTRL  )
                                                     OR   (BRPOT_CNCL_SPD_PRGM_SWH  AND PORT_CTRL_EOT)(* SPEED OVERRIDE    PORT     *)
                                                     OR   ( BRSTBD_CNCL_SPD_PRGM_SWH  AND  STBD_CTRL_EOT    )(* SPEED OVERRIDE     STBD     *)
                                                     OR  CRASH_REVERSE_SPEEDPROGRAMOVERRIDE
                                                     OR  (BR_CNCEL_SPEED_PRGM_LMP_INTERNAL AND BR_CTRL)
                                                     OR (ECR_CNCEL_SPD_PRGM_LMP_INTERNAL AND ECRA_CTRL) ;




(* CANCEL  LIMITS   *)
CANCEL_LIMITS_BX:=(CANCEL_LIMITS_BR AND  BR_CTRL)
                                          OR  (CANCEL_LIMITS_ECRA AND  ECRA_CTRL)
                                          OR ( BRPOT_CANCEL_LIMIT_SWH  AND  PORT_CTRL_EOT ) (* CANCEL  LIMITS      PORT  *)
                                          OR(  BRSTBD_CANCEL_LIMIT_SWH  AND  STBD_CTRL_EOT) (* CANCEL  LIMITS      STBD  *)
                                          OR CRASH_REVERSE_CANCELL_LIMITS
                                          OR (BR_CNCL_LIMIT_LMP_INTERNAL AND BR_CTRL)
                                          OR (ECR_CNCEL_LIMIT_LMP_INTERNAL AND ECRA_CTRL);




(*-------------UNIC  SPEED  CONTROLLER  FEEDBACK------------*)
H_SPEED_PRGM_ACTIVE:= SPEED_PRGM_ACTIVE_INDIC;


H_SPD_PRGM_OVERD:=SPEED_OVERD_INDIC_BX;


H_ENG_OUTPUT_LIMITED:=ENG_OUTPUT_LIMITED_BX;


H_SETPOINT_CRITICAL_SPD_BX:=SETPOINT_CRITICAL_SPD_BX;


H_ENG_CRITICAL_SPD_BX:=ENG_CRITICAL_SPD_BX;
END_FUNCTION_BLOCK

(* POU LAMP_TEST, ST *)
FUNCTION_BLOCK LAMP_TEST
VAR_INPUT
END_VAR
VAR_OUTPUT
END_VAR
VAR



END_VAR
(* ---------------------- LAMP TEST-------------------------------*)
BR_ECR_PUBSH_ALARM_TEST:=BR_LAMP_TEST_PB_INTERNAL OR ECR_LAMP_TEST_PB_INTERNAL OR PORT_LAMP_TEST_PB_INTERNAL OR STBD_LAMP_TEST_PB_INTERNAL ;

IF ALRM_ACKSOUND_OFF_BR
THEN
	 H_HORN_ALARM_BRG:=FALSE ;
END_IF;

IF ALRM_ACKSOUND_OFF_ECR
THEN
       H_HORN_ALARM_ECR:=FALSE ;
END_IF;

IF ALRM_ACKSOUND_OFF_PORT
THEN
	 H_HORN_ALARM_BRG:=FALSE ;
END_IF;

IF ALRM_ACKSOUND_OFF_STBD
THEN
		 H_HORN_ALARM_BRG:=FALSE ;
END_IF;

(* -----------------------------------ACOUSTIC    SIGNALS ---------------------------------*)
    ENG_FAIL_ACOUSTIC :=  HornStartInterlock  OR startFail OR SlowTurnFailBX;
END_FUNCTION_BLOCK

(* POU LAMP, ST *)
FUNCTION_BLOCK LAMP
VAR_INPUT
END_VAR
VAR

	FLAG: BOOL;
	FLAG_BR_LMT: BOOL;
	FLAG_ECRA_LMT: BOOL;
	FLAG_POT_LMT: BOOL;
	FLAG_STBD_LMT: BOOL;
	FLAG_PRGM_BR: BOOL;
	FLAG_PRGM_ECA: BOOL;
	FLAG_PRGM_PRGM: BOOL;
	FLAG_STBD_PRGM: BOOL;

END_VAR
VAR_IN_OUT

END_VAR
IF (CANCEL_LIMITS_BR AND (NOT FLAG_BR_LMT))
THEN
         BR_CNCL_LIMIT_LMP_INTERNAL:=NOT BR_CNCL_LIMIT_LMP_INTERNAL;
          FLAG_BR_LMT:=TRUE;
END_IF;
IF( NOT CANCEL_LIMITS_BR)
THEN
         FLAG_BR_LMT:=FALSE;
END_IF;



IF (CANCEL_LIMITS_ECRA  AND (NOT FLAG_ECRA_LMT))
THEN
       ECR_CNCEL_LIMIT_LMP_INTERNAL:=NOT  ECR_CNCEL_LIMIT_LMP_INTERNAL   ;
       FLAG_ECRA_LMT:=TRUE;
END_IF
IF(  NOT CANCEL_LIMITS_ECRA )
THEN
        FLAG_ECRA_LMT:=FALSE;
END_IF;

IF (BRPOT_CANCEL_LIMIT_SWH AND (NOT FLAG_POT_LMT))
THEN
	BR_PORT_CNCEL_LIMIT_LMP_INTERNAL:=NOT BR_PORT_CNCEL_LIMIT_LMP_INTERNAL ;
        FLAG_POT_LMT:=TRUE;
END_IF
IF(NOT BRPOT_CANCEL_LIMIT_SWH)
THEN
          FLAG_POT_LMT:=FALSE;
END_IF;


IF (BRSTBD_CANCEL_LIMIT_SWH AND (NOT FLAG_STBD_LMT))
THEN
      BR_STBD_CNCEL_LIMIT_LMP_INTERNAL:=NOT  BR_STBD_CNCEL_LIMIT_LMP_INTERNAL;
     FLAG_STBD_LMT:=TRUE;
END_IF;
IF(NOT  BRSTBD_CANCEL_LIMIT_SWH)
THEN
       FLAG_STBD_LMT:=FALSE;
END_IF;


IF ( SPEED_PRGM_OVERRIDE_BR AND  (NOT FLAG_PRGM_BR))
THEN
	BR_CNCEL_SPEED_PRGM_LMP_INTERNAL:=NOT BR_CNCEL_SPEED_PRGM_LMP_INTERNAL;
       FLAG_PRGM_BR:=TRUE;
END_IF
IF(NOT SPEED_PRGM_OVERRIDE_BR)
THEN
     FLAG_PRGM_BR:=FALSE;
END_IF


IF (SPEED_PRGM_OVERRIDE_ECA AND  ( NOT FLAG_PRGM_ECA))
THEN
	ECR_CNCEL_SPD_PRGM_LMP_INTERNAL:= NOT ECR_CNCEL_SPD_PRGM_LMP_INTERNAL;
      FLAG_PRGM_ECA:=TRUE;
END_IF
IF( NOT SPEED_PRGM_OVERRIDE_ECA)
THEN
  FLAG_PRGM_ECA:=FALSE;
END_IF;

IF (BRPOT_CNCL_SPD_PRGM_SWH AND ( NOT  FLAG_PRGM_PRGM))
THEN
	BR_PORT_CNCEL_SPD_PRGM_LMP_INTERNAL:=NOT BR_PORT_CNCEL_SPD_PRGM_LMP_INTERNAL ;
        FLAG_PRGM_PRGM:=TRUE;
END_IF
IF( NOT BRPOT_CNCL_SPD_PRGM_SWH)
THEN
           FLAG_PRGM_PRGM:=FALSE;
END_IF

IF (BRSTBD_CNCL_SPD_PRGM_SWH AND FLAG=FALSE)
THEN
	BR_STBD_CNCEL_SPD_PRGM_LMP_INTERNAL:= NOT  BR_STBD_CNCEL_SPD_PRGM_LMP_INTERNAL;
       FLAG_STBD_PRGM:=TRUE;
END_IF
IF (NOT BRSTBD_CNCL_SPD_PRGM_SWH)
THEN
          FLAG_STBD_PRGM:=FALSE;
END_IF
END_FUNCTION_BLOCK

(* POU PARAM_HW, ST *)
FUNCTION_BLOCK PARAM_HW
VAR_INPUT
END_VAR
VAR_OUTPUT
END_VAR
VAR
	SPEED_TO_WATCH_INST:SPEED_TO_WATCH;


	FLAG: BOOL;
END_VAR
(*---------------HW   Signal list-------------------*)

(*----------------------------------------AI----------------------------------------*)
 HW_ANALOG_SPEED_RCS:=WORD_TO_INT(HW_ANALOG_SPEED_RCS_HW);(*PRORCST5101C*)
 POSITION_HIGHWORD:=RCS_Engine_Speed1A_HIG ;(* PRORCST5102C  FI*)
 POSITION_LOWWORD:=RCS_Engine_Speed1B_LOW;(*PRORCST5103C  FI*)
  MVL_POSITION_BR:=WORD_TO_REAL(BR_MVL_COMMD);       (*PRORCS1001  *)
  MVL_POSITION_ECR:=WORD_TO_REAL(ECR_MVL_COMMD);(*PRORCS1002*)
(*----------------------------------------AO----------------------------------------*)
 SPEED_TO_WATCH_INST(RCS_SPEED_VALUE:=RCS_SPEED_MEANSURE_VALUE);
  BR_ENGINE_SPEED_METER1 :=INT_TO_WORD(SPEED_TO_WATCH_INST.VALUE); (*PRORCS1003*)
  BR_ENGINE_SPEED_METER2  := INT_TO_WORD( SPEED_TO_WATCH_INST.VALUE); (*PRORCS1004*)
  BR_ENGINE_SPEED_METER3  :=INT_TO_WORD( SPEED_TO_WATCH_INST.VALUE);(*PRORCS1005*)
  BR_ENGINE_SPEED_METER  :=INT_TO_WORD( SPEED_TO_WATCH_INST.VALUE);  (*PRORCS1006*)
  BR_PORT_WING_ENGINE_SPEED_METER  :=INT_TO_WORD( SPEED_TO_WATCH_INST.VALUE); (*PRORCS1007*)
  BR_STBD_WING_ENGINE_SPEED_METER   :=INT_TO_WORD( SPEED_TO_WATCH_INST.VALUE); (*PRORCS1008*)
  CHIEF_RM_ENGINE_SPEED_METER   :=INT_TO_WORD( SPEED_TO_WATCH_INST.VALUE); (*PRORCS1009*)
  BR_START_AIR_PRESS_METER:=REAL_TO_WORD( StartAirPress);(*PRORCS1010*)
  BR_PORT_WING_START_AIR_PRESS_METER:=REAL_TO_WORD( StartAirPress);(*PRORCS1011*)
  BR_STBD_WING_START_AIR_PRESS_METER:=REAL_TO_WORD( StartAirPress);(*PRORCS1012*)
  ECR_START_AIR_PRESS_METER:=REAL_TO_WORD( StartAirPress);(*PRORCS1013*)
  FUEL_LOAD_INDEX:=REAL_TO_WORD(Estimated_Engine_Load_Internal);(*PRORCS1055*)

(*----------------------------------------DI----------------------------------------*)
  RCS_HW_overspd:=RCS_OVERSPEED_HW;(*PRORCS1014*)
  BR_PUS_BR_CTRL:=BR_BRIDGE_APPLY_FOR_CONTROL;(*PRORCS1015*)
  BR_PUS_ECRA_CTRL:=BR_ECR_AUTO_APPLY_FOR_CONTROL AND BRG_ECRA_CTRL_FLSH;  (*PRORCS1016*)
  BR_PUS_ECRM_CTRL:=BR_ECR_AUTO_APPLY_FOR_CONTROL AND BRG_ECRM_CTRL_FLSH;  (*PRORCS1016*)
  BR_PUS_LOC_MAN_CTRL:=BR_LOCAL_MAN_APPLY_FOR_CONTROL;(*PRORCS1017*)
  BR_LAMP_TEST_PB_INTERNAL:=BR_LAMP_TEST_PB;(*PRORCS1018*)
  ECRA_PUS_BR_CTRL:=ECR_BRIDGE_APPLY_FOR_CONTROL;(*PRORCS1020*)
  ECRA_PUS_ECRA_CTRL:=ECR_ECR_AUTO_APPLY_FOR_CONTROL; (*PRORCS1021*)
  ECRA_PUS_LOC_MAN_CTRL:=ECR_LOCAL_MAN_APPLY_FOR_CONTROL;(*PRORCS1022*)
 PlantInterlock:=PLANT_REALERLOCK;(*PRORCS1023*)
 ECR_LAMP_TEST_PB_INTERNAL:=ECR_LAMP_TEST_PB; (*PRORCS1024*)
 SafetyStop:=SAFETY_STOP OR  safety_stop_mb ;(* PRORCS1026   SAFETY_STOP come  from HW    Safety_STOP_MB  come  from modbus*)
 SafetySystemOff:=NOT SAFETY_SYSTEM_OFF_HW;(*PRORCS1027---------------------Safety is ready =true------------NOT READY ->START INTERLOCK*)
 SAFETY_SYSTEM_OFF_FAIL:=SAFETY_SYSTEM_OFF_FAIL_HW;(*PRORCS1085 *)
 PORT_LAMP_TEST_PB_INTERNAL:=PORT_LAMP_TEST_PB;(*PRORCS1028*)
 STBD_LAMP_TEST_PB_INTERNAL:=STBD_LAMP_TEST_PB;(*PRORCS1030*)
  CANCEL_LIMITS_BR:=BR_CANCEL_LIMIT_SWH_HW;(*PRORCS1057*)
  SPEED_PRGM_OVERRIDE_BR:= BR_CNCL_SPD_PRGM_SWH_HW;(*PRORCS1058*)

  CANCEL_LIMITS_ECRA:=ECRA_CANCEL_LIMIT_SWH_HW;(*PRORCS1059*)
  SPEED_PRGM_OVERRIDE_ECA:=ECRA_CNCL_SPD_PRGM_SWH_HW;(*PRORCS1060*)
  BRPOT_CANCEL_LIMIT_SWH:=BRPOT_CANCEL_LIMIT_SWH_HW;(*PRORCS1061*)
  BRPOT_CNCL_SPD_PRGM_SWH:=BRPOT_CNCL_SPD_PRGM_SWH_HW;(*PRORCS1062*)
  BRSTBD_CANCEL_LIMIT_SWH:=BRSTBD_CANCEL_LIMIT_SWH_HW;(*PRORCS1063*)
  BRSTBD_CNCL_SPD_PRGM_SWH:=BRSTBD_CNCL_SPD_PRGM_SWH_HW;(*PRORCS1064*)
  PORT_CTRL_EOT:=PORT_CTRL_EOT_HW;(*PRORCS1076*)
  STBD_CTRL_EOT:=STBD_CTRL_EOT_HW;(*PRORCS1077*)
  SLOW_DOWN:=SLOW_DOWN_HW;(*PRORCS1080*)
  PCS_POWER_SUPPLY_ALM:=PCS_POWER_SUPPLY_ALM_HW;(*   PRORCS1041*)

(*----------------------------------------DO----------------------------------------*)
(*BR_LAMP_TEST_PB_INTERNAL  IS   TESTBED  BUTTON*)

 BR_BRIDGE_IN_CONTROL:=BR_LAMPS_BR_CTRL OR BR_LAMP_TEST_PB_INTERNAL ;(*PRORCS1032*)
 BR_ECR_AUTO_MAN_IN_CONTROL:=BR_LAMPS_ECRA_CTRL  OR BR_LAMPS_ECRM_CTRL OR BR_LAMP_TEST_PB_INTERNAL ;(*PRORCS1033 *)
 BR_LOCAL_MAN_IN_CONTROL:= BR_LAMPS_LOCAL_MAN_CTRL  OR BR_LAMP_TEST_PB_INTERNAL  ;(*PRORCS1034*)

BR_LAMP_TEST_INDICATOR:=BR_LAMP_TEST_PB_INTERNAL   ;(*PRORCS1035*)


ECR_BRIDGE_IN_CONTROL:=ECR_LAMPS_BR_CTRL   OR ECR_LAMP_TEST_PB_INTERNAL;(* PRORCS1038*)
ECR_ECR_AUTO_IN_CONTROL:=ECR_LAMPS_ECRA_CTRL   OR ECR_LAMP_TEST_PB_INTERNAL;(*PRORCS1039*)
ECR_LOCAL_MAN_IN_CONTROL:=ECR_LAMPS_LOCAL_MAN_CTRL   OR ECR_LAMP_TEST_PB_INTERNAL;(*PRORCS1040*)

ECT_LAMP_TEST_INDICATOR:=ECR_LAMP_TEST_PB_INTERNAL ;(*PRORCS1042*)

PORT_LAMP_TEST_INDICATOR:=   PORT_LAMP_TEST_PB_INTERNAL ;(*PRORCS1049*)
STBD_LAMP_TEST_INDICATOR:=STBD_LAMP_TEST_INDICATOR_INTERNAL;(*PRORCS1052*)

(*WRONG_WAY_ALARM_ECR:=WRONG_WAY_ALARM;(*PRORCS1044*)-----------DELETE*)
REVOLUTION_COUNTER_INDICATOR:=REVOLUTION_COUNTER_PULSE;(*PRORCS1045*)
(* WRONG_WAY_ALARM_LOCAL:=WRONG_WAY_ALARM;(*PRORCS1046*)-----------DELETE*)
ECR_BRIDGE_IN_CONTROL_EOT:=ECR_BRIDGE_IN_CONTROL_INTERNAL;(*PRORCS1047*)
ECR_ECR_AUTO_IN_CONTROL_EOT:=ECR_ECR_AUTO_IN_CONTROL_INTERNAL;(*PRORCS1048*)
(*BR_PORT_WRONG_WAY_ALARM  :=WRONG_WAY_ALARM;(*PRORCS1051*)-----------DELETE*)
(*BR_STBD_WRONG_WAY_ALARM :=WRONG_WAY_ALARM;(*PRORCS1054*)-----------DELETE*)
Propulsion_Control_Failure_ALM:= propulsion_ctrl_failure_alm;(*PRORCXS9001A*)
Propulsion_Control_Passive_Failure_ALM:=propulsion_ctrl_passive_failure_alm;(*PRORCXS9002A*)
PCS_ENG_Speed_Meas_Failure_ALM:=PCS_SPD_MEASURE_FAILURE;(*PRORCXS9003A*)
Engine_Standstill_RUN_STOPPED:=EngineStandstill;(*PRORCXS9005A*)
RUNNING_HOUR_INIDICATOR:=ENG_RUNING_HRS;(*PRORCS1056*)


IF  (NOT   BR_CNCL_LIMIT_LMP_INTERNAL)
THEN   BR_CNCEL_LIMIT_LMP_HW:=(OUTPUT_LIMIT_FLASHER AND BR_CTRL) OR BR_LAMP_TEST_PB_INTERNAL ; (*PRORCS1065*)
ELSE   BR_CNCEL_LIMIT_LMP_HW:=  (BR_CNCL_LIMIT_LMP_INTERNAL AND BR_CTRL) OR BR_LAMP_TEST_PB_INTERNAL ;(*PRORCS1065*)
END_IF;

IF ( NOT ECR_CNCEL_LIMIT_LMP_INTERNAL )
THEN ECR_CNCEL_LIMIT_LMP_HW:=(OUTPUT_LIMIT_FLASHER AND ECRA_CTRL) OR ECR_LAMP_TEST_PB_INTERNAL;(*PRORCS1067*)
ELSE  ECR_CNCEL_LIMIT_LMP_HW:=(ECR_CNCEL_LIMIT_LMP_INTERNAL AND ECRA_CTRL) OR ECR_LAMP_TEST_PB_INTERNAL;(*PRORCS1067*)
END_IF;

IF (NOT  BR_CNCEL_SPEED_PRGM_LMP_INTERNAL)
THEN  BR_CNCEL_SPEED_PRGM_LMP_HW:=(SPEED_PRO_FLASHER AND BR_CTRL) OR BR_LAMP_TEST_PB_INTERNAL ;(*PRORCS1066*)
ELSE   BR_CNCEL_SPEED_PRGM_LMP_HW:=(BR_CNCEL_SPEED_PRGM_LMP_INTERNAL AND BR_CTRL) OR BR_LAMP_TEST_PB_INTERNAL ;(*PRORCS1066*)
END_IF;

IF (NOT  ECR_CNCEL_SPD_PRGM_LMP_INTERNAL)
THEN   ECR_CNCEL_SPD_PRGM_LMP_HW:=(SPEED_PRO_FLASHER AND ECRA_CTRL) OR ECR_LAMP_TEST_PB_INTERNAL;(*PRORCS1068*)
ELSE   ECR_CNCEL_SPD_PRGM_LMP_HW:=(ECR_CNCEL_SPD_PRGM_LMP_INTERNAL AND ECRA_CTRL) OR ECR_LAMP_TEST_PB_INTERNAL;(*PRORCS1068*)
END_IF;

BR_PORT_CNCEL_LIMIT_LMP_HW:=(BR_PORT_CNCEL_LIMIT_LMP_INTERNAL AND BR_CTRL ) OR PORT_LAMP_TEST_PB_INTERNAL  ;(*PRORCS1069*)
BR_PORT_CNCEL_SPD_PRGM_LMP_HW:=(BR_PORT_CNCEL_SPD_PRGM_LMP_INTERNAL AND BR_CTRL) OR PORT_LAMP_TEST_PB_INTERNAL ;(*PRORCS1070*)

BR_STBD_CNCEL_LIMIT_LMP_HW:=(BR_STBD_CNCEL_LIMIT_LMP_INTERNAL AND BR_CTRL) OR STBD_LAMP_TEST_PB_INTERNAL  ;(*PRORCS1071*)
BR_STBD_CNCEL_SPD_PRGM_LMP_HW:=(BR_STBD_CNCEL_SPD_PRGM_LMP_INTERNAL AND BR_CTRL) OR STBD_LAMP_TEST_PB_INTERNAL ;(*PRORCS1072*)



H_WRONG_WAY_ALARM:=WRONG_WAY_ALARM;
END_FUNCTION_BLOCK

(* POU Speed_TO_Watch, ST *)
FUNCTION_BLOCK Speed_TO_Watch
VAR_INPUT
	RCS_SPEED_VALUE:REAL;
END_VAR
VAR_OUTPUT
	VALUE:INT;
END_VAR
VAR
	K_VALUE: REAL;
	B_VALUE: REAL;
END_VAR
K_VALUE:=(SPEED_AO_MAX  -  SPEED_AO_MIN)/300;
B_VALUE:=SPEED_AO_MAX-150*K_VALUE;

IF  EngTurningAST
THEN  RCS_SPEED_VALUE:=-RCS_SPEED_VALUE;
END_IF;

VALUE:=REAL_TO_INT(RCS_SPEED_VALUE*K_VALUE+B_VALUE);
END_FUNCTION_BLOCK

(* POU PARAM_MODBUS, ST *)
FUNCTION_BLOCK PARAM_MODBUS
VAR
	flag: INT;
END_VAR
   MODBUS_CONFIGURATION;
   IF  MBCFG_ESS.MBCFG_Error=MBCFG_NO_Error THEN
   alrm_acksound_off_br_mb:= MBCFG_ESS.alrm_acksound_off_br_cfg;(* ESS:   PROESS0118 	%QX274.1*)
   alrm_acksound_off_ecr_mb:=MBCFG_ESS.alrm_acksound_off_ecr_cfg;(* ESS:   PROESS0119  	%QX274.2*)
   alrm_acksound_off_port_mb:=MBCFG_ESS.alrm_acksound_off_port_cfg;(* ESS:  PROESS0120	%QX274.3*)
   alrm_acksound_off_stbd_mb:=MBCFG_ESS.alrm_acksound_off_stbd_cfg;(* ESS:  PROESS0121	%QX274.4*)
   ess_eng_speed_bkp_mb:=MBCFG_ESS.ess_eng_speed_bkp_cfg;(*ESS: PROESS0004	%QW256*)
   ess_eng_standstill_bkp_mb:=MBCFG_ESS.ess_eng_standstill_bkp_cfg;(*ESS: PROESS0003   %QX270.0*)
   ess_eng_turning_ahead_bkp_mb:=MBCFG_ESS.ess_eng_turning_ahead_bkp_cfg;(* ESS: PROESS0072  %QX272.0 *)
   ess_eng_turning_astern_bkp_mb:=MBCFG_ESS.ess_eng_turning_astern_bkp_cfg;(*ESS: PROESS0073  %QX272.1*)
   ess_overspeed_sw_bkp_mb:=MBCFG_ESS.ess_overspeed_sw_bkp_cfg;(*ESS: PROESS0062   %QX271.11 *)
   ess_overspeed_hw_bkp_mb:=MBCFG_ESS.ess_overspeed_hw_bkp_cfg;(*ESS: PROESS0075   %QX272.2 *)
   (*safety_system_off_mb:=MBCFG_ESS.safety_system_off_cfg;(*ESS:  PROESS0103  %QX274.0*)-----DELETE*)
   safety_stop_mb:=MBCFG_ESS.safety_stop_cfg;(*ESS:  PROESS0065 %QX271.13 *)
    ess_can_communicationLost:=MBCFG_ESS.ess_can_communicationLost_cfg;
ELSE
  alrm_acksound_off_br_mb:= MBCFG_ESS_2.alrm_acksound_off_br_cfg;(* ESS:   PROESS0118 	%QX274.1*)
   alrm_acksound_off_ecr_mb:=MBCFG_ESS_2.alrm_acksound_off_ecr_cfg;(* ESS:   PROESS0119  	%QX274.2*)
   alrm_acksound_off_port_mb:=MBCFG_ESS_2.alrm_acksound_off_port_cfg;(* ESS:  PROESS0120	%QX274.3*)
   alrm_acksound_off_stbd_mb:=MBCFG_ESS_2.alrm_acksound_off_stbd_cfg;(* ESS:  PROESS0121	%QX274.4*)
   ess_eng_speed_bkp_mb:=MBCFG_ESS_2.ess_eng_speed_bkp_cfg;(*ESS: PROESS0004	%QW256*)
   ess_eng_standstill_bkp_mb:=MBCFG_ESS_2.ess_eng_standstill_bkp_cfg;(*ESS: PROESS0003   %QX270.0*)
   ess_eng_turning_ahead_bkp_mb:=MBCFG_ESS_2.ess_eng_turning_ahead_bkp_cfg;(* ESS: PROESS0072  %QX272.0 *)
   ess_eng_turning_astern_bkp_mb:=MBCFG_ESS_2.ess_eng_turning_astern_bkp_cfg;(*ESS: PROESS0073  %QX272.1*)
   ess_overspeed_sw_bkp_mb:=MBCFG_ESS_2.ess_overspeed_sw_bkp_cfg;(*ESS: PROESS0062   %QX271.11 *)
   ess_overspeed_hw_bkp_mb:=MBCFG_ESS_2.ess_overspeed_hw_bkp_cfg;(*ESS: PROESS0075   %QX272.2 *)
   (*safety_system_off_mb:=MBCFG_ESS.safety_system_off_cfg;(*ESS:  PROESS0103  %QX274.0*)-----DELETE*)
   safety_stop_mb:=MBCFG_ESS_2.safety_stop_cfg;(*ESS:  PROESS0065 %QX271.13 *)
    ess_can_communicationLost:=MBCFG_ESS_2.ess_can_communicationLost_cfg;

   END_IF;

(*------------------------------------------------------------MODBUS INPUT----------------------------------------------------------------------*)
IF(SPT_no_gearteeth_per_rev>0)
THEN
      AllowRestartResetDelay:=REAL_TO_TIME(SPT_al_restar_reset_dly)*1000;    (* al_restar_reset_dly  :REAL; SEC->mSEC*)

	CHIEFLIMIT:=SPT_chief_limit;           (*chief_limit  :REAL*)

	CrashMovDly:=REAL_TO_TIME(SPT_crash_ast_mov_dly)*1000;  (*crash_ast_mov_dly	:REAL SEC->mSEC*)

	Enable_Crash_Astern_S1:=SPT_crash_ast_mvl_abv_lim; (*crash_ast_mvl_abv_lim	:REAL*)

	Activate_Crash_Astern_S2:=SPT_crash_ast_mvl_bel_lim;  (*crash_ast_mvl_bel_lim	:REAL*)

	Real_Crash_Astern_S3:=SPT_crash_ast_rst_spd_lim;    (*crash_ast_rst_spd_lim	:REAL*)

       EngineRuningDelay:=REAL_TO_TIME(SPT_eng_running_dly)*1000	;(*eng_running_dly	AT	:REAL*)

      STANDSTILL_SETPOINT:=REAL_TO_INT(SPT_engine_standstill);   (*  engine_standstill	AT	%IW270	:REAL*)

      SPEED_FACTOR_B:=SPT_fac_b_for_eng_spd;(*REAL_TO_INT(SPT_fac_b_for_eng_spd);   (*fac_b_for_eng_spd	AT	%IW272	:REAL*)*)

	SPEED_FACTOR_C:=SPT_fac_c_for_eng_spd;(*REAL_TO_INT(SPT_fac_c_for_eng_spd) ;  (*fac_c_for_eng_spd	AT	%IW274	:REAL*)*)

       HZ:= SPT_flash_frequency  ;   (*    flash_frequency	AT	%IW276	:REAL*)

	LO_CHIEF_LIMIT:=SPT_lo_chief_imit	;(*lo_chief_imit	AT	%IW278	:REAL*)

	MAX_SPEED:=SPT_max_speed_mb ;(*max_speed	AT	%IW280	:REAL*)

      GRADE_RPM_ELEC_MAP[4].RPM:=SPT_mvl_dslow_ahd_sp;(*mvl_dslow_ahd_sp	AT	%IW282	:REAL*)

      GRADE_RPM_ELEC_MAP[6].RPM:=SPT_mvl_dslow_ast_sp;(*mvl_dslow_ast_sp	AT	%IW284	:REAL*)

      GRADE_RPM_ELEC_MAP[1].RPM:=SPT_mvl_ful_ahd_sp;(*mvl_ful_ahd_sp	AT	%IW286	:REAL*)

      GRADE_RPM_ELEC_MAP[0].RPM:=SPT_mvl_ful_sea_ahd_sp;(*mvl_ful_sea_ahd_sp	AT	%IW288	:REAL*)

      GRADE_RPM_ELEC_MAP[9].RPM:=SPT_mvl_full_ast_sp;(* mvl_full_ast_sp	AT	%IW290	:REAL *)

      GRADE_RPM_ELEC_MAP[10].RPM:=SPT_mvl_full_sea_ast_sp;(*mvl_full_sea_ast_sp	AT	%IW292	:REAL  *)

      GRADE_RPM_ELEC_MAP[2].RPM:=SPT_mvl_half_ahd_sp;(*mvl_half_ahd_sp	AT	%IW294	:REAL*)

      GRADE_RPM_ELEC_MAP[8].RPM:=SPT_mvl_half_ast_sp;(*mvl_half_ast_sp	AT	%IW296	:REAL*)

      MVL_HANDLE_MATCH:=SPT_mvl_hand_match_thld*ConvertValue ;(*mvl_hand_match_thld	AT	%IW298	:REAL ConvertValue:=1638=1mA  *)

      MVL_POS_AHEAD_VALUE:=SPT_mvl_posi_ahead_val*ConvertValue	;(*  mvl_posi_ahead_val	AT	%IW300	:REAL*)

      MVL_POS_ASTERN_VALUE:=SPT_mvl_posi_astern_val*ConvertValue;(* mvl_posi_astern_val	AT	%IW302	:REAL ConvertValue:=1638=1mA*)

     GRADE_RPM_ELEC_MAP[3].RPM:=SPT_mvl_slow_ahd_sp;(* mvl_slow_ahd_sp	AT	%IW304	:REAL *)

     GRADE_RPM_ELEC_MAP[7].RPM:=SPT_mvl_slow_ast_sp;(* mvl_slow_ast_sp	AT	%IW306	:REAL *)

     GRADE_RPM_ELEC_MAP[5].RPM:=SPT_mvl_stop;(*mvl_stop	AT	%IW308	:REAL  *)

     NBreakHIGH:= SPT_n_brake_thld_hi;(*n_brake_thld_hi	AT	%IW310	:REAL*)

     NStartLOW:=SPT_n_start_thld_lo;(*n_start_thld_lo	AT	%IW312	:REAL*)

     NStartHIGH:=SPT_n_start_thld_hi;(*n_start_thld_hi	AT	%ID285	:REAL;*)

     NBreakLOW:=SPT_n_brake_thld_lo;(*n_brake_thld_lo	AT	%IW316	:REAL*)

     GEAR_TEETH_PER_REVOLUTION_SETPOINT:=REAL_TO_INT(SPT_no_gearteeth_per_rev);(*no_gearteeth_per_rev	AT	%IW318	:REAL*)

     RATE_OF_CHANGE_FAST:=SPT_rate_chan_fast	;(*rate_chan_fast	AT	%IW320	:REAL*)

     RATE_OF_CHANGE_SLOW:=SPT_rate_chan_low;(*rate_chan_low	AT	%IW322	:REAL*)

     RstartInhibitDelay:=REAL_TO_TIME(SPT_restar_inhibit_dly)*1000;(*restar_inhibit_dly	AT	%IW324	:REAL    SEC->mSEC*)

    REVOLUTION_COUNTER_FACTOR_SETPOINT:=REAL_TO_INT(SPT_rev_count_factor);(*SPT_rev_count_factor	AT	%IW326	:REAL *)

    SLOW_DOWN_VALUE:= SPT_slowdown_val;(*slowdown_val	AT	%IW328	:REAL*)

     IF(SPT_slowturn_by_MVL_enab=1) (*slowturn_by_MVL_enab	AT	%IW330	:REAL*)
    THEN  SlowByMVLEnable:=TRUE;
    ELSE   SlowByMVLEnable:=FALSE;
    END_IF

    SlowTurnDelayRequest:=REAL_TO_TIME(SPT_slowturn_del_req)*60*1000;(*slowturn_del_req	AT	%IW332	:REAL        MIN->MSEC*)

     SPEED_CMCR:=SPT_spd_CMCR;(* 	SPT_spd_CMCR AT %IW334 : REAL;*)

    PULSE_TIME:=REAL_TO_TIME(SPT_spd_pulse_time)*1000 ;(*spd_pulse_time	AT	%IW336	:REAL   SEC->mSEC*)

    StartAirPreHIGH :=SPT_star_air_pres_hi	;(*star_air_pres_hi	AT	%IW338	:REAL*)

    StartAirPreLow:=SPT_star_air_pres_low	;(*star_air_pres_low	AT	%IW340	:REAL*)

    SPD_SIM_MODE_ACTIVE:=SPT_sim_mode_active;(*SPT_sim_mode_active AT %QW344 : REAL;*)

    SMI_SPD_FROM_HMI:=SPT_speed_from_hmi;(*SPT_speed_from_hmi AT %QW346 : REAL;*)

    SIMULATION_TARGET_VALUE_FROMHMI :=SPT_speed_hmi;(*SPT_speed_hmi AT %QW348 : REAL; *)

    OVERSPEED_SETPOINT:=REAL_TO_INT(SPT_over_speed);(*SPT_over_speed AT %QW342 : REAL;*)

    ess_engine_turning_ahead_bkp:=  ess_eng_turning_ahead_bkp_mb OR  ESS_ENG_TURN_AHD_BKP_HW ;(*ModBus OR  HW----------------------ENG..AHEAD*)

    ess_engine_turning_astern_bkp:=ess_eng_turning_astern_bkp_mb  OR   ESS_ENG_TURN_AST_BKP_HW ;(*ModBus OR  HW-----------------------ENG  ASTERN*)

    ess_engine_standstill_bakup:=ess_eng_standstill_bkp_mb;

    ess_overspeed_sw_bakup:=ess_overspeed_sw_bkp_mb;

   ess_overspeed_hw_bakup:=ess_overspeed_hw_bkp_mb;

   ALRM_ACKSOUND_OFF_BR:=alrm_acksound_off_br_mb;

   ALRM_ACKSOUND_OFF_ECR:=alrm_acksound_off_ecr_mb;

   ALRM_ACKSOUND_OFF_PORT:=alrm_acksound_off_port_mb;

   ALRM_ACKSOUND_OFF_STBD:=alrm_acksound_off_stbd_mb;

   (*SafetySystemOff:=safety_system_off_mb OR SAFETY_SYSTEM_OFF_HW ; MOVE HW*)
     eng_speed_setpoint_rc:=SPEED_SETPOINT_BX;  (*PRORCS0090     eng_speed_setpoint_rc     %QW264;*)

      Critical_Speed_Enable:= SPT_Critical_Speed_Enable ;

      Critical_RPM_low1:=	SPT_Critical_RPM_low1 ;

	Critical_RPM_high1:=SPT_Critical_RPM_high1;

	Critical_RPM_low2:=SPT_Critical_RPM_low2;

      Critical_RPM_high2:=SPT_Critical_RPM_high2 ;

END_IF;



(*---------------------------------MODBUS     OUTPUT  TO  HMI---------------------------------*)

	start_air_pressure:=StartAirPress/100 ;                             (*PRORCCAN0001  start_air_pressure            %QW256*)

    (*  eng_revolution_counter  AT  %QW258:  REAL;*)    (*PRORCS0055     eng_revolution_counter      %QW258*)

    (*  eng_running_hours:=ENG_RUNING_HRS;           (*PRORCS0056     eng_running_hours  AT       %QW260*)------------DELETE*)

	rcs_eng_speed1:=NPN_DETECT_SPEED_RCS;   (*PRORCS0089     rcs_eng_speed1                 %QW262:*)


	eng_speed_setpoint_rc:=SPEED_SETPOINT_BX; (*PRORCS0090     eng_speed_setpoint_rc     %QW264;*)

	fuel_index:=Estimated_Engine_Load_Internal*0.1;       (*PRORCS0104     engine Load                              %QW466*)

    h_fuel_index:=Fuel_Index_can*0.1; (*PRORCS7174, fuel _index *)

